Yaskawa INFORM job: DEMO_ROOF_UPPER_0625_3PAINT_8.JBI

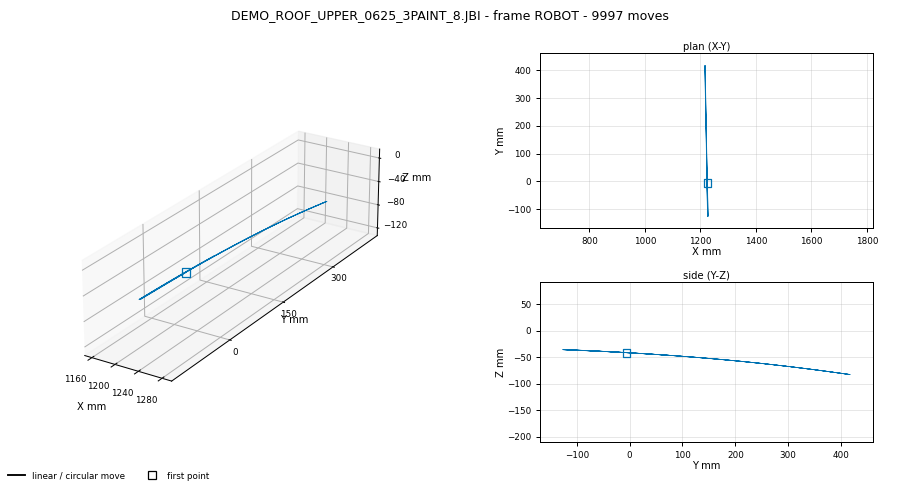
[picture p0: tool path of DEMO_ROOF_UPPER_0625_3PAINT_8.JBI in frame ROBOT, 9997 of 9997 moves have a stored position in this frame; points joined in program order, loops and branches not executed]
/JOB
//NAME DEMO_ROOF_UPPER_0625_3PAINT8
//POS
///NPOS 9997,0,0,0,0,0
///TOOL 0
///USER 0
///POSTYPE ROBOT
///RECTAN
///RCONF 1,0,0,0,0,0,0,0,0,0,0,0,0,0,0,0,0,0,0,0,0,0,0,0
C00000=1225.284,-6.004,-41.147,-179.569,5.363,148.803
C00001=1225.289,-6.253,-41.132,-179.571,5.363,148.804
C00002=1225.293,-6.503,-41.118,-179.574,5.362,148.805
C00003=1225.298,-6.753,-41.104,-179.576,5.362,148.805
C00004=1225.303,-7.002,-41.089,-179.579,5.361,148.806
C00005=1225.308,-7.251,-41.076,-179.581,5.362,148.807
C00006=1225.313,-7.501,-41.063,-179.584,5.361,148.807
C00007=1225.318,-7.751,-41.048,-179.586,5.361,148.808
C00008=1225.323,-8.001,-41.034,-179.588,5.361,148.809
C00009=1225.329,-8.250,-41.020,-179.591,5.360,148.809
C00010=1225.334,-8.500,-41.006,-179.594,5.360,148.810
C00011=1225.339,-8.749,-40.992,-179.596,5.359,148.811
C00012=1225.344,-8.999,-40.977,-179.598,5.360,148.811
C00013=1225.349,-9.248,-40.964,-179.601,5.359,148.812
C00014=1225.354,-9.497,-40.950,-179.604,5.359,148.813
C00015=1225.359,-9.747,-40.935,-179.606,5.359,148.814
C00016=1225.364,-9.997,-40.922,-179.609,5.358,148.814
C00017=1225.369,-10.246,-40.908,-179.611,5.358,148.815
C00018=1225.374,-10.496,-40.894,-179.614,5.357,148.816
C00019=1225.379,-10.746,-40.880,-179.616,5.358,148.816
C00020=1225.384,-10.995,-40.866,-179.619,5.357,148.817
C00021=1225.389,-11.244,-40.852,-179.621,5.357,148.818
C00022=1225.394,-11.495,-40.838,-179.623,5.357,148.818
C00023=1225.400,-11.744,-40.824,-179.625,5.356,148.819
C00024=1225.405,-11.993,-40.810,-179.628,5.356,148.820
C00025=1225.409,-12.243,-40.796,-179.630,5.356,148.820
C00026=1225.414,-12.492,-40.782,-179.633,5.355,148.821
C00027=1225.420,-12.742,-40.769,-179.636,5.355,148.822
C00028=1225.425,-12.992,-40.755,-179.638,5.354,148.822
C00029=1225.429,-13.241,-40.741,-179.640,5.355,148.823
C00030=1225.435,-13.490,-40.727,-179.643,5.354,148.824
C00031=1225.440,-13.741,-40.713,-179.646,5.354,148.824
C00032=1225.445,-13.990,-40.699,-179.648,5.354,148.825
C00033=1225.450,-14.239,-40.686,-179.650,5.353,148.826
C00034=1225.455,-14.489,-40.672,-179.653,5.353,148.826
C00035=1225.460,-14.739,-40.658,-179.655,5.353,148.827
C00036=1225.465,-14.988,-40.644,-179.658,5.353,148.828
C00037=1225.470,-15.237,-40.630,-179.660,5.352,148.829
C00038=1225.475,-15.487,-40.617,-179.663,5.352,148.829
C00039=1225.480,-15.737,-40.603,-179.665,5.352,148.830
C00040=1225.485,-15.986,-40.589,-179.668,5.352,148.831
C00041=1225.490,-16.236,-40.576,-179.670,5.351,148.831
C00042=1225.495,-16.485,-40.562,-179.672,5.351,148.832
C00043=1225.500,-16.735,-40.548,-179.675,5.351,148.833
C00044=1225.506,-16.985,-40.535,-179.678,5.350,148.833
C00045=1225.510,-17.234,-40.521,-179.680,5.351,148.834
C00046=1225.516,-17.484,-40.507,-179.683,5.350,148.835
C00047=1225.521,-17.733,-40.494,-179.685,5.350,148.835
C00048=1225.526,-17.983,-40.480,-179.687,5.350,148.836
C00049=1225.531,-18.233,-40.466,-179.690,5.349,148.837
C00050=1225.536,-18.482,-40.452,-179.693,5.349,148.838
C00051=1225.541,-18.732,-40.439,-179.695,5.350,148.838
C00052=1225.546,-18.981,-40.425,-179.698,5.349,148.839
C00053=1225.551,-19.231,-40.411,-179.700,5.349,148.840
C00054=1225.556,-19.480,-40.398,-179.703,5.349,148.841
C00055=1225.561,-19.730,-40.384,-179.705,5.348,148.841
C00056=1225.567,-19.979,-40.371,-179.708,5.348,148.842
C00057=1225.572,-20.229,-40.357,-179.710,5.348,148.843
C00058=1225.577,-20.479,-40.344,-179.713,5.348,148.843
C00059=1225.582,-20.728,-40.330,-179.715,5.347,148.844
C00060=1225.587,-20.978,-40.317,-179.717,5.347,148.845
C00061=1225.592,-21.227,-40.303,-179.720,5.347,148.845
C00062=1225.597,-21.477,-40.290,-179.723,5.346,148.846
C00063=1225.602,-21.726,-40.276,-179.725,5.346,148.847
C00064=1225.607,-21.977,-40.263,-179.727,5.346,148.848
C00065=1225.612,-22.246,-40.248,-179.730,5.346,148.848
C00066=1225.618,-22.515,-40.233,-179.733,5.345,148.849
C00067=1225.624,-22.784,-40.218,-179.735,5.345,148.850
C00068=1225.629,-23.054,-40.205,-179.738,5.345,148.851
C00069=1225.634,-23.303,-40.191,-179.741,5.345,148.851
C00070=1225.639,-23.553,-40.178,-179.743,5.344,148.852
C00071=1225.645,-23.802,-40.164,-179.745,5.345,148.853
C00072=1225.649,-24.052,-40.151,-179.748,5.344,148.853
C00073=1225.654,-24.302,-40.137,-179.751,5.344,148.854
C00074=1225.659,-24.551,-40.124,-179.753,5.344,148.855
C00075=1225.664,-24.801,-40.110,-179.755,5.344,148.855
C00076=1225.670,-25.050,-40.097,-179.758,5.343,148.856
C00077=1225.674,-25.300,-40.084,-179.760,5.343,148.857
C00078=1225.680,-25.550,-40.070,-179.763,5.343,148.857
C00079=1225.685,-25.799,-40.057,-179.766,5.342,148.858
C00080=1225.690,-26.049,-40.044,-179.768,5.343,148.859
C00081=1225.695,-26.298,-40.030,-179.770,5.342,148.860
C00082=1225.701,-26.548,-40.017,-179.773,5.342,148.860
C00083=1225.705,-26.798,-40.004,-179.775,5.342,148.861
C00084=1225.710,-27.047,-39.990,-179.778,5.342,148.862
C00085=1225.716,-27.296,-39.977,-179.780,5.341,148.862
C00086=1225.720,-27.546,-39.964,-179.782,5.341,148.863
C00087=1225.726,-27.795,-39.950,-179.785,5.341,148.864
C00088=1225.730,-28.045,-39.937,-179.788,5.340,148.864
C00089=1225.736,-28.295,-39.924,-179.790,5.341,148.865
C00090=1225.741,-28.545,-39.911,-179.792,5.340,148.866
C00091=1225.746,-28.794,-39.897,-179.795,5.340,148.867
C00092=1225.751,-29.044,-39.884,-179.797,5.340,148.867
C00093=1225.757,-29.294,-39.871,-179.800,5.339,148.868
C00094=1225.761,-29.543,-39.857,-179.802,5.340,148.869
C00095=1225.766,-29.792,-39.845,-179.805,5.339,148.869
C00096=1225.772,-30.042,-39.832,-179.807,5.339,148.870
C00097=1225.776,-30.292,-39.819,-179.809,5.339,148.871
C00098=1225.782,-30.541,-39.805,-179.812,5.339,148.871
C00099=1225.786,-30.791,-39.792,-179.815,5.338,148.872
C00100=1225.792,-31.040,-39.779,-179.817,5.338,148.873
C00101=1225.797,-31.291,-39.766,-179.819,5.338,148.874
C00102=1225.802,-31.540,-39.753,-179.822,5.337,148.874
C00103=1225.808,-31.789,-39.739,-179.824,5.338,148.875
C00104=1225.812,-32.039,-39.726,-179.827,5.337,148.876
C00105=1225.817,-32.288,-39.714,-179.829,5.338,148.876
C00106=1225.822,-32.539,-39.700,-179.832,5.337,148.877
C00107=1225.828,-32.788,-39.687,-179.834,5.337,148.878
C00108=1225.833,-33.037,-39.675,-179.836,5.337,148.878
C00109=1225.838,-33.287,-39.660,-179.839,5.336,148.879
C00110=1225.843,-33.536,-39.648,-179.842,5.336,148.880
C00111=1225.847,-33.786,-39.635,-179.844,5.336,148.881
C00112=1225.853,-34.036,-39.622,-179.846,5.336,148.881
C00113=1225.858,-34.285,-39.609,-179.848,5.336,148.882
C00114=1225.863,-34.535,-39.596,-179.851,5.336,148.883
C00115=1225.869,-34.785,-39.583,-179.854,5.335,148.883
C00116=1225.874,-35.034,-39.570,-179.856,5.335,148.884
C00117=1225.878,-35.284,-39.557,-179.859,5.335,148.885
C00118=1225.884,-35.533,-39.543,-179.861,5.334,148.885
C00119=1225.888,-35.783,-39.530,-179.863,5.335,148.886
C00120=1225.893,-36.033,-39.518,-179.866,5.334,148.887
C00121=1225.899,-36.282,-39.505,-179.869,5.334,148.888
C00122=1225.904,-36.532,-39.492,-179.871,5.334,148.888
C00123=1225.909,-36.782,-39.479,-179.873,5.334,148.889
C00124=1225.914,-37.031,-39.467,-179.875,5.334,148.890
C00125=1225.919,-37.281,-39.453,-179.878,5.333,148.890
C00126=1225.924,-37.531,-39.440,-179.881,5.333,148.891
C00127=1225.930,-37.780,-39.428,-179.883,5.333,148.892
C00128=1225.934,-38.030,-39.415,-179.885,5.333,148.892
C00129=1225.940,-38.280,-39.402,-179.888,5.333,148.893
C00130=1225.945,-38.529,-39.389,-179.890,5.333,148.894
C00131=1225.950,-38.779,-39.376,-179.893,5.332,148.895
C00132=1225.955,-39.028,-39.363,-179.895,5.332,148.895
C00133=1225.961,-39.278,-39.350,-179.898,5.332,148.896
C00134=1225.966,-39.527,-39.338,-179.900,5.331,148.897
C00135=1225.970,-39.777,-39.325,-179.902,5.332,148.897
C00136=1225.975,-40.026,-39.312,-179.905,5.331,148.898
C00137=1225.981,-40.276,-39.299,-179.907,5.332,148.899
C00138=1225.986,-40.526,-39.286,-179.910,5.331,148.899
C00139=1225.991,-40.775,-39.273,-179.912,5.331,148.900
C00140=1225.996,-41.025,-39.261,-179.915,5.331,148.901
C00141=1226.001,-41.275,-39.248,-179.917,5.330,148.902
C00142=1226.006,-41.525,-39.236,-179.919,5.331,148.902
C00143=1226.011,-41.774,-39.223,-179.922,5.330,148.903
C00144=1226.017,-42.024,-39.210,-179.925,5.330,148.904
C00145=1226.021,-42.274,-39.197,-179.927,5.330,148.904
C00146=1226.027,-42.523,-39.184,-179.929,5.330,148.905
C00147=1226.032,-42.772,-39.172,-179.931,5.330,148.906
C00148=1226.037,-43.022,-39.159,-179.934,5.329,148.906
C00149=1226.041,-43.272,-39.146,-179.937,5.329,148.907
C00150=1226.047,-43.522,-39.134,-179.939,5.329,148.908
C00151=1226.053,-43.771,-39.121,-179.942,5.329,148.909
C00152=1226.058,-44.020,-39.109,-179.944,5.328,148.909
C00153=1226.062,-44.271,-39.096,-179.946,5.329,148.910
C00154=1226.067,-44.520,-39.083,-179.949,5.328,148.911
C00155=1226.073,-44.769,-39.070,-179.951,5.329,148.911
C00156=1226.078,-45.019,-39.059,-179.954,5.328,148.912
C00157=1226.083,-45.269,-39.046,-179.956,5.328,148.913
C00158=1226.088,-45.518,-39.033,-179.958,5.328,148.913
C00159=1226.093,-45.768,-39.020,-179.961,5.327,148.914
C00160=1226.099,-46.017,-39.007,-179.963,5.328,148.915
C00161=1226.104,-46.267,-38.995,-179.966,5.327,148.916
C00162=1226.109,-46.517,-38.982,-179.968,5.328,148.916
C00163=1226.114,-46.767,-38.970,-179.971,5.327,148.917
C00164=1226.119,-47.016,-38.957,-179.973,5.327,148.918
C00165=1226.124,-47.266,-38.945,-179.975,5.327,148.918
C00166=1226.129,-47.515,-38.933,-179.978,5.326,148.919
C00167=1226.134,-47.765,-38.920,-179.980,5.327,148.920
C00168=1226.139,-48.015,-38.907,-179.983,5.326,148.920
C00169=1226.145,-48.284,-38.895,-179.986,5.326,148.921
C00170=1226.151,-48.554,-38.880,-179.988,5.327,148.922
C00171=1226.156,-48.825,-38.867,-179.991,5.326,148.923
C00172=1226.162,-49.094,-38.854,-179.993,5.326,148.923
C00173=1226.166,-49.344,-38.841,-179.996,5.325,148.924
C00174=1226.172,-49.594,-38.829,-179.998,5.325,148.925
C00175=1226.177,-49.843,-38.817,179.999,5.325,148.926
C00176=1226.182,-50.092,-38.804,179.997,5.325,148.926
C00177=1226.187,-50.342,-38.792,179.994,5.325,148.927
C00178=1226.192,-50.591,-38.779,179.992,5.325,148.928
C00179=1226.197,-50.841,-38.766,179.990,5.325,148.928
C00180=1226.202,-51.091,-38.755,179.987,5.324,148.929
C00181=1226.207,-51.341,-38.742,179.985,5.324,148.930
C00182=1226.213,-51.590,-38.729,179.982,5.324,148.931
C00183=1226.218,-51.840,-38.717,179.980,5.324,148.931
C00184=1226.223,-52.089,-38.705,179.978,5.324,148.932
C00185=1226.229,-52.339,-38.693,179.975,5.323,148.933
C00186=1226.234,-52.589,-38.680,179.973,5.324,148.933
C00187=1226.238,-52.839,-38.667,179.970,5.323,148.934
C00188=1226.244,-53.089,-38.656,179.968,5.324,148.935
C00189=1226.249,-53.338,-38.643,179.965,5.323,148.935
C00190=1226.254,-53.588,-38.631,179.963,5.323,148.936
C00191=1226.259,-53.837,-38.619,179.961,5.323,148.937
C00192=1226.264,-54.087,-38.607,179.958,5.322,148.938
C00193=1226.269,-54.336,-38.595,179.956,5.323,148.938
C00194=1226.275,-54.586,-38.583,179.953,5.322,148.939
C00195=1226.279,-54.836,-38.570,179.951,5.323,148.940
C00196=1226.284,-55.086,-38.558,179.948,5.322,148.940
C00197=1226.290,-55.335,-38.545,179.946,5.322,148.941
C00198=1226.295,-55.585,-38.533,179.944,5.322,148.942
C00199=1226.300,-55.834,-38.521,179.941,5.322,148.942
C00200=1226.305,-56.084,-38.509,179.939,5.322,148.943
C00201=1226.310,-56.333,-38.497,179.936,5.321,148.944
C00202=1226.315,-56.583,-38.485,179.934,5.322,148.945
C00203=1226.321,-56.833,-38.472,179.932,5.321,148.945
C00204=1226.326,-57.083,-38.460,179.929,5.322,148.946
C00205=1226.331,-57.332,-38.448,179.927,5.321,148.947
C00206=1226.336,-57.582,-38.437,179.924,5.321,148.947
C00207=1226.341,-57.831,-38.424,179.922,5.321,148.948
C00208=1226.346,-58.081,-38.412,179.919,5.321,148.949
C00209=1226.351,-58.331,-38.399,179.917,5.321,148.950
C00210=1226.356,-58.581,-38.387,179.915,5.320,148.950
C00211=1226.362,-58.831,-38.375,179.913,5.321,148.951
C00212=1226.366,-59.080,-38.363,179.910,5.320,148.952
C00213=1226.372,-59.330,-38.351,179.908,5.321,148.952
C00214=1226.377,-59.579,-38.339,179.905,5.320,148.953
C00215=1226.382,-59.829,-38.327,179.902,5.320,148.954
C00216=1226.388,-60.079,-38.315,179.900,5.320,148.954
C00217=1226.392,-60.328,-38.303,179.898,5.320,148.955
C00218=1226.397,-60.578,-38.291,179.896,5.320,148.956
C00219=1226.403,-60.828,-38.279,179.893,5.319,148.957
C00220=1226.408,-61.077,-38.267,179.891,5.320,148.957
C00221=1226.413,-61.327,-38.255,179.888,5.319,148.958
C00222=1226.418,-61.577,-38.244,179.885,5.319,148.959
C00223=1226.423,-61.826,-38.231,179.883,5.319,148.959
C00224=1226.429,-62.076,-38.219,179.881,5.319,148.960
C00225=1226.433,-62.325,-38.208,179.879,5.319,148.961
C00226=1226.438,-62.575,-38.195,179.876,5.319,148.962
C00227=1226.444,-62.825,-38.183,179.874,5.319,148.962
C00228=1226.449,-63.075,-38.171,179.871,5.318,148.963
C00229=1226.454,-63.324,-38.160,179.869,5.319,148.964
C00230=1226.459,-63.574,-38.148,179.866,5.318,148.964
C00231=1226.464,-63.824,-38.136,179.864,5.318,148.965
C00232=1226.469,-64.073,-38.124,179.862,5.318,148.966
C00233=1226.474,-64.322,-38.112,179.859,5.318,148.966
C00234=1226.480,-64.572,-38.100,179.857,5.318,148.967
C00235=1226.485,-64.822,-38.088,179.854,5.318,148.968
C00236=1226.490,-65.072,-38.077,179.852,5.318,148.969
C00237=1226.495,-65.322,-38.065,179.850,5.317,148.969
C00238=1226.501,-65.571,-38.053,179.847,5.318,148.970
C00239=1226.506,-65.820,-38.041,179.845,5.317,148.971
C00240=1226.511,-66.070,-38.029,179.843,5.318,148.971
C00241=1226.517,-66.320,-38.017,179.840,5.317,148.972
C00242=1226.521,-66.570,-38.006,179.837,5.317,148.973
C00243=1226.526,-66.819,-37.994,179.835,5.317,148.974
C00244=1226.532,-67.069,-37.982,179.833,5.317,148.974
C00245=1226.536,-67.319,-37.970,179.830,5.317,148.975
C00246=1226.542,-67.568,-37.959,179.828,5.316,148.976
C00247=1226.547,-67.818,-37.947,179.826,5.317,148.976
C00248=1226.552,-68.068,-37.935,179.823,5.316,148.977
C00249=1226.557,-68.317,-37.923,179.821,5.317,148.978
C00250=1226.562,-68.567,-37.911,179.818,5.316,148.978
C00251=1226.568,-68.816,-37.900,179.816,5.317,148.979
C00252=1226.573,-69.066,-37.888,179.814,5.316,148.980
C00253=1226.578,-69.316,-37.877,179.811,5.316,148.981
C00254=1226.583,-69.566,-37.865,179.809,5.316,148.981
C00255=1226.588,-69.815,-37.854,179.806,5.315,148.982
C00256=1226.594,-70.065,-37.842,179.804,5.316,148.983
C00257=1226.599,-70.315,-37.830,179.801,5.315,148.983
C00258=1226.604,-70.565,-37.819,179.799,5.316,148.984
C00259=1226.609,-70.814,-37.806,179.797,5.315,148.985
C00260=1226.614,-71.063,-37.795,179.795,5.316,148.986
C00261=1226.620,-71.313,-37.783,179.792,5.315,148.986
C00262=1226.624,-71.563,-37.772,179.790,5.315,148.987
C00263=1226.630,-71.813,-37.760,179.787,5.315,148.988
C00264=1226.634,-72.062,-37.749,179.785,5.315,148.988
C00265=1226.640,-72.312,-37.737,179.782,5.315,148.989
C00266=1226.645,-72.562,-37.725,179.780,5.315,148.990
C00267=1226.650,-72.811,-37.714,179.778,5.315,148.991
C00268=1226.656,-73.061,-37.702,179.775,5.314,148.991
C00269=1226.661,-73.311,-37.691,179.773,5.315,148.992
C00270=1226.666,-73.561,-37.679,179.770,5.314,148.993
C00271=1226.671,-73.810,-37.668,179.768,5.315,148.993
C00272=1226.676,-74.060,-37.656,179.765,5.314,148.994
C00273=1226.682,-74.330,-37.644,179.763,5.314,148.995
C00274=1226.688,-74.601,-37.631,179.761,5.314,148.995
C00275=1226.693,-74.871,-37.620,179.758,5.314,148.996
C00276=1226.698,-75.141,-37.607,179.755,5.314,148.997
C00277=1226.704,-75.391,-37.595,179.753,5.314,148.998
C00278=1226.709,-75.641,-37.583,179.751,5.314,148.999
C00279=1226.714,-75.891,-37.572,179.748,5.314,148.999
C00280=1226.719,-76.139,-37.561,179.746,5.314,149.000
C00281=1226.725,-76.390,-37.549,179.743,5.314,149.001
C00282=1226.730,-76.640,-37.538,179.741,5.314,149.001
C00283=1226.735,-76.890,-37.526,179.738,5.313,149.002
C00284=1226.740,-77.138,-37.515,179.736,5.314,149.003
C00285=1226.746,-77.388,-37.503,179.734,5.313,149.003
C00286=1226.751,-77.638,-37.492,179.732,5.313,149.004
C00287=1226.755,-77.888,-37.481,179.729,5.313,149.005
C00288=1226.761,-78.138,-37.469,179.727,5.312,149.005
C00289=1226.766,-78.387,-37.458,179.725,5.313,149.006
C00290=1226.772,-78.637,-37.447,179.722,5.312,149.007
C00291=1226.776,-78.887,-37.436,179.720,5.313,149.008
C00292=1226.782,-79.137,-37.424,179.717,5.312,149.008
C00293=1226.787,-79.386,-37.413,179.715,5.313,149.009
C00294=1226.792,-79.635,-37.402,179.712,5.312,149.010
C00295=1226.798,-79.886,-37.390,179.710,5.312,149.010
C00296=1226.802,-80.135,-37.379,179.708,5.312,149.011
C00297=1226.808,-80.384,-37.368,179.706,5.312,149.012
C00298=1226.813,-80.634,-37.356,179.703,5.312,149.012
C00299=1226.818,-80.884,-37.345,179.701,5.312,149.013
C00300=1226.823,-81.134,-37.334,179.698,5.312,149.014
C00301=1226.829,-81.383,-37.323,179.696,5.312,149.015
C00302=1226.833,-81.633,-37.312,179.693,5.312,149.015
C00303=1226.839,-81.883,-37.300,179.691,5.312,149.016
C00304=1226.844,-82.133,-37.289,179.689,5.312,149.017
C00305=1226.849,-82.382,-37.278,179.687,5.312,149.017
C00306=1226.855,-82.632,-37.266,179.684,5.311,149.018
C00307=1226.859,-82.882,-37.255,179.682,5.312,149.019
C00308=1226.864,-83.132,-37.244,179.679,5.311,149.020
C00309=1226.870,-83.381,-37.233,179.677,5.312,149.020
C00310=1226.875,-83.631,-37.222,179.674,5.311,149.021
C00311=1226.880,-83.880,-37.210,179.672,5.312,149.022
C00312=1226.885,-84.130,-37.200,179.670,5.311,149.022
C00313=1226.891,-84.380,-37.188,179.667,5.312,149.023
C00314=1226.895,-84.629,-37.177,179.665,5.311,149.024
C00315=1226.901,-84.879,-37.167,179.663,5.311,149.024
C00316=1226.906,-85.129,-37.155,179.661,5.311,149.025
C00317=1226.911,-85.379,-37.144,179.658,5.311,149.026
C00318=1226.916,-85.629,-37.133,179.656,5.311,149.026
C00319=1226.921,-85.878,-37.122,179.654,5.311,149.027
C00320=1226.927,-86.128,-37.110,179.651,5.310,149.028
C00321=1226.932,-86.378,-37.100,179.649,5.311,149.029
C00322=1226.937,-86.627,-37.089,179.646,5.310,149.029
C00323=1226.942,-86.877,-37.078,179.644,5.311,149.030
C00324=1226.948,-87.127,-37.066,179.641,5.310,149.031
C00325=1226.953,-87.376,-37.055,179.639,5.311,149.031
C00326=1226.958,-87.626,-37.045,179.637,5.310,149.032
C00327=1226.963,-87.876,-37.033,179.635,5.310,149.033
C00328=1226.969,-88.126,-37.023,179.632,5.310,149.034
C00329=1226.974,-88.375,-37.011,179.630,5.310,149.034
C00330=1226.979,-88.624,-37.000,179.627,5.310,149.035
C00331=1226.984,-88.874,-36.990,179.625,5.310,149.036
C00332=1226.989,-89.124,-36.979,179.622,5.310,149.036
C00333=1226.995,-89.374,-36.968,179.620,5.310,149.037
C00334=1227.000,-89.624,-36.956,179.618,5.310,149.038
C00335=1227.005,-89.874,-36.946,179.616,5.310,149.038
C00336=1227.010,-90.123,-36.935,179.613,5.309,149.039
C00337=1227.015,-90.373,-36.924,179.611,5.310,149.040
C00338=1227.021,-90.622,-36.913,179.609,5.309,149.040
C00339=1227.026,-90.872,-36.902,179.607,5.310,149.041
C00340=1227.031,-91.122,-36.891,179.604,5.309,149.042
C00341=1227.036,-91.372,-36.881,179.602,5.309,149.043
C00342=1227.041,-91.621,-36.870,179.599,5.309,149.043
C00343=1227.046,-91.871,-36.859,179.597,5.309,149.044
C00344=1227.051,-92.120,-36.848,179.594,5.309,149.045
C00345=1227.057,-92.371,-36.837,179.592,5.309,149.045
C00346=1227.062,-92.620,-36.826,179.590,5.309,149.046
C00347=1227.067,-92.870,-36.815,179.587,5.309,149.047
C00348=1227.072,-93.119,-36.804,179.585,5.309,149.048
C00349=1227.077,-93.369,-36.794,179.583,5.309,149.048
C00350=1227.082,-93.619,-36.783,179.580,5.309,149.049
C00351=1227.088,-93.869,-36.772,179.578,5.309,149.050
C00352=1227.093,-94.119,-36.762,179.576,5.308,149.050
C00353=1227.099,-94.368,-36.750,179.574,5.309,149.051
C00354=1227.104,-94.618,-36.740,179.571,5.308,149.052
C00355=1227.109,-94.867,-36.729,179.569,5.309,149.052
C00356=1227.114,-95.117,-36.718,179.566,5.308,149.053
C00357=1227.120,-95.367,-36.708,179.564,5.308,149.054
C00358=1227.124,-95.617,-36.697,179.561,5.308,149.054
C00359=1227.129,-95.867,-36.686,179.559,5.308,149.055
C00360=1227.135,-96.116,-36.675,179.557,5.308,149.056
C00361=1227.140,-96.366,-36.665,179.555,5.308,149.057
C00362=1227.145,-96.616,-36.654,179.552,5.308,149.057
C00363=1227.150,-96.865,-36.643,179.550,5.308,149.058
C00364=1227.156,-97.115,-36.633,179.547,5.308,149.059
C00365=1227.161,-97.365,-36.622,179.545,5.308,149.059
C00366=1227.166,-97.614,-36.611,179.543,5.307,149.060
C00367=1227.172,-97.864,-36.600,179.541,5.308,149.061
C00368=1227.177,-98.114,-36.590,179.538,5.307,149.061
C00369=1227.182,-98.364,-36.579,179.536,5.308,149.062
C00370=1227.187,-98.613,-36.569,179.534,5.308,149.063
C00371=1227.192,-98.863,-36.558,179.531,5.307,149.063
C00372=1227.198,-99.113,-36.548,179.529,5.308,149.064
C00373=1227.203,-99.363,-36.536,179.526,5.307,149.065
C00374=1227.208,-99.612,-36.526,179.524,5.308,149.066
C00375=1227.213,-99.862,-36.516,179.522,5.307,149.066
C00376=1227.219,-100.111,-36.505,179.520,5.308,149.067
C00377=1227.224,-100.383,-36.494,179.517,5.307,149.068
C00378=1227.230,-100.654,-36.482,179.514,5.307,149.068
C00379=1227.235,-100.924,-36.471,179.512,5.307,149.069
C00380=1227.241,-101.196,-36.459,179.509,5.307,149.070
C00381=1227.247,-101.445,-36.449,179.507,5.307,149.071
C00382=1227.251,-101.695,-36.438,179.505,5.307,149.071
C00383=1227.257,-101.944,-36.428,179.503,5.307,149.072
C00384=1227.262,-102.195,-36.417,179.500,5.307,149.073
C00385=1227.267,-102.444,-36.408,179.498,5.307,149.073
C00386=1227.272,-102.694,-36.397,179.495,5.307,149.074
C00387=1227.277,-102.943,-36.386,179.493,5.307,149.075
C00388=1227.282,-103.193,-36.376,179.490,5.306,149.076
C00389=1227.288,-103.443,-36.365,179.488,5.307,149.076
C00390=1227.293,-103.693,-36.355,179.486,5.306,149.077
C00391=1227.298,-103.943,-36.345,179.484,5.306,149.078
C00392=1227.304,-104.192,-36.334,179.482,5.307,149.078
C00393=1227.309,-104.442,-36.324,179.479,5.306,149.079
C00394=1227.314,-104.691,-36.313,179.477,5.307,149.080
C00395=1227.319,-104.942,-36.302,179.474,5.306,149.080
C00396=1227.324,-105.191,-36.293,179.472,5.307,149.081
C00397=1227.329,-105.441,-36.282,179.470,5.306,149.082
C00398=1227.335,-105.691,-36.272,179.468,5.307,149.083
C00399=1227.340,-105.940,-36.262,179.465,5.306,149.083
C00400=1227.345,-106.190,-36.251,179.463,5.306,149.084
C00401=1227.351,-106.440,-36.241,179.461,5.306,149.084
C00402=1227.356,-106.690,-36.230,179.459,5.306,149.085
C00403=1227.361,-106.940,-36.220,179.456,5.306,149.086
C00404=1227.366,-107.188,-36.210,179.454,5.306,149.087
C00405=1227.371,-107.439,-36.199,179.451,5.306,149.087
C00406=1227.377,-107.688,-36.189,179.449,5.306,149.088
C00407=1227.382,-107.938,-36.178,179.446,5.305,149.089
C00408=1227.387,-108.188,-36.168,179.444,5.306,149.089
C00409=1227.393,-108.437,-36.158,179.442,5.306,149.090
C00410=1227.397,-108.687,-36.148,179.440,5.305,149.091
C00411=1227.403,-108.937,-36.138,179.438,5.306,149.091
C00412=1227.408,-109.187,-36.128,179.435,5.305,149.092
C00413=1227.413,-109.437,-36.117,179.433,5.306,149.093
C00414=1227.419,-109.686,-36.107,179.430,5.305,149.094
C00415=1227.423,-109.936,-36.097,179.428,5.306,149.094
C00416=1227.429,-110.186,-36.087,179.426,5.305,149.095
C00417=1227.434,-110.435,-36.076,179.424,5.306,149.096
C00418=1227.439,-110.686,-36.066,179.421,5.305,149.096
C00419=1227.445,-110.935,-36.056,179.419,5.305,149.097
C00420=1227.450,-111.184,-36.046,179.417,5.305,149.098
C00421=1227.455,-111.435,-36.035,179.415,5.305,149.098
C00422=1227.460,-111.684,-36.025,179.412,5.305,149.099
C00423=1227.466,-111.934,-36.015,179.410,5.305,149.100
C00424=1227.471,-112.184,-36.006,179.408,5.305,149.100
C00425=1227.476,-112.434,-35.996,179.405,5.305,149.101
C00426=1227.482,-112.683,-35.985,179.403,5.305,149.102
C00427=1227.487,-112.934,-35.975,179.400,5.305,149.103
C00428=1227.492,-113.183,-35.965,179.399,5.305,149.103
C00429=1227.497,-113.432,-35.955,179.396,5.304,149.104
C00430=1227.502,-113.683,-35.944,179.394,5.305,149.104
C00431=1227.508,-113.932,-35.934,179.391,5.304,149.105
C00432=1227.513,-114.181,-35.925,179.389,5.305,149.106
C00433=1227.518,-114.431,-35.914,179.386,5.304,149.107
C00434=1227.524,-114.682,-35.904,179.384,5.305,149.107
C00435=1227.528,-114.931,-35.895,179.382,5.305,149.108
C00436=1227.534,-115.181,-35.885,179.380,5.304,149.109
C00437=1227.539,-115.431,-35.874,179.378,5.305,149.109
C00438=1227.544,-115.680,-35.864,179.375,5.304,149.110
C00439=1227.549,-115.930,-35.854,179.373,5.305,149.111
C00440=1227.555,-116.180,-35.845,179.370,5.304,149.111
C00441=1227.560,-116.430,-35.835,179.368,5.305,149.112
C00442=1227.565,-116.679,-35.825,179.366,5.304,149.113
C00443=1227.571,-116.929,-35.814,179.364,5.304,149.113
C00444=1227.576,-117.178,-35.805,179.361,5.304,149.114
C00445=1227.581,-117.429,-35.795,179.359,5.304,149.115
C00446=1227.587,-117.678,-35.785,179.357,5.304,149.115
C00447=1227.591,-117.928,-35.775,179.355,5.304,149.116
C00448=1227.596,-118.178,-35.764,179.352,5.304,149.117
C00449=1227.602,-118.427,-35.754,179.350,5.304,149.118
C00450=1227.607,-118.677,-35.745,179.348,5.304,149.118
C00451=1227.613,-118.927,-35.735,179.346,5.304,149.119
C00452=1227.618,-119.176,-35.725,179.343,5.304,149.120
C00453=1227.623,-119.426,-35.715,179.341,5.304,149.120
C00454=1227.629,-119.676,-35.705,179.339,5.304,149.121
C00455=1227.633,-119.926,-35.696,179.336,5.303,149.122
C00456=1227.639,-120.175,-35.686,179.334,5.304,149.122
C00457=1227.644,-120.426,-35.676,179.332,5.304,149.123
C00458=1227.649,-120.675,-35.666,179.330,5.303,149.124
C00459=1227.655,-120.925,-35.656,179.328,5.304,149.124
C00460=1227.660,-121.174,-35.646,179.325,5.303,149.125
C00461=1227.666,-121.424,-35.637,179.323,5.304,149.126
C00462=1227.670,-121.674,-35.627,179.320,5.303,149.126
C00463=1227.675,-121.924,-35.617,179.318,5.304,149.127
C00464=1227.681,-122.174,-35.607,179.316,5.303,149.128
C00465=1227.686,-122.423,-35.598,179.314,5.303,149.128
C00466=1227.691,-122.673,-35.587,179.312,5.304,149.129
C00467=1227.696,-122.923,-35.578,179.309,5.303,149.130
C00468=1227.702,-123.173,-35.568,179.307,5.304,149.131
C00469=1227.707,-123.422,-35.558,179.304,5.303,149.131
C00470=1227.713,-123.672,-35.549,179.303,5.303,149.132
C00471=1227.718,-123.921,-35.539,179.300,5.303,149.132
C00472=1227.723,-124.172,-35.529,179.298,5.303,149.133
C00473=1227.728,-124.421,-35.520,179.295,5.303,149.134
C00474=1227.733,-124.671,-35.509,179.293,5.303,149.135
C00475=1227.739,-124.921,-35.501,179.290,5.303,149.135
C00476=1227.744,-125.170,-35.490,179.289,5.303,149.136
C00477=1227.749,-125.420,-35.481,179.287,5.303,149.137
C00478=1227.754,-125.671,-35.471,179.284,5.303,149.137
C00479=1227.759,-125.920,-35.462,179.282,5.303,149.138
C00480=1227.765,-126.170,-35.452,179.279,5.303,149.139
C00481=1227.343,-126.181,-35.488,179.275,5.306,149.141
C00482=1227.338,-125.931,-35.497,179.277,5.307,149.140
C00483=1227.333,-125.681,-35.507,179.279,5.306,149.139
C00484=1227.328,-125.431,-35.517,179.282,5.307,149.139
C00485=1227.322,-125.181,-35.527,179.284,5.306,149.138
C00486=1227.317,-124.932,-35.536,179.286,5.306,149.137
C00487=1227.312,-124.682,-35.546,179.289,5.306,149.137
C00488=1227.307,-124.433,-35.555,179.291,5.306,149.136
C00489=1227.301,-124.182,-35.565,179.293,5.307,149.135
C00490=1227.296,-123.933,-35.575,179.295,5.306,149.135
C00491=1227.291,-123.683,-35.585,179.298,5.307,149.134
C00492=1227.286,-123.433,-35.594,179.300,5.306,149.133
C00493=1227.280,-123.184,-35.604,179.303,5.307,149.132
C00494=1227.275,-122.934,-35.613,179.304,5.307,149.132
C00495=1227.269,-122.684,-35.623,179.307,5.306,149.131
C00496=1227.264,-122.434,-35.634,179.309,5.307,149.131
C00497=1227.259,-122.184,-35.643,179.311,5.306,149.130
C00498=1227.254,-121.934,-35.653,179.314,5.307,149.129
C00499=1227.249,-121.685,-35.663,179.316,5.306,149.128
C00500=1227.243,-121.435,-35.672,179.318,5.307,149.128
C00501=1227.239,-121.185,-35.682,179.320,5.307,149.127
C00502=1227.233,-120.936,-35.692,179.323,5.307,149.126
C00503=1227.228,-120.686,-35.701,179.325,5.307,149.126
C00504=1227.222,-120.436,-35.711,179.328,5.307,149.125
C00505=1227.217,-120.187,-35.722,179.330,5.307,149.124
C00506=1227.212,-119.937,-35.732,179.332,5.307,149.124
C00507=1227.207,-119.687,-35.741,179.334,5.307,149.123
C00508=1227.202,-119.437,-35.751,179.336,5.307,149.122
C00509=1227.196,-119.188,-35.761,179.339,5.307,149.122
C00510=1227.191,-118.937,-35.771,179.341,5.307,149.121
C00511=1227.186,-118.688,-35.780,179.344,5.308,149.120
C00512=1227.180,-118.438,-35.791,179.346,5.307,149.120
C00513=1227.175,-118.189,-35.801,179.349,5.308,149.119
C00514=1227.170,-117.938,-35.810,179.350,5.308,149.118
C00515=1227.165,-117.689,-35.820,179.352,5.307,149.118
C00516=1227.160,-117.439,-35.830,179.355,5.308,149.117
C00517=1227.154,-117.190,-35.840,179.357,5.307,149.116
C00518=1227.149,-116.939,-35.851,179.360,5.308,149.115
C00519=1227.144,-116.690,-35.860,179.362,5.307,149.115
C00520=1227.138,-116.440,-35.870,179.364,5.308,149.114
C00521=1227.133,-116.191,-35.880,179.366,5.308,149.114
C00522=1227.128,-115.941,-35.890,179.369,5.308,149.113
C00523=1227.123,-115.691,-35.900,179.371,5.308,149.112
C00524=1227.117,-115.441,-35.910,179.373,5.308,149.111
C00525=1227.113,-115.191,-35.920,179.376,5.308,149.111
C00526=1227.107,-114.941,-35.930,179.378,5.308,149.110
C00527=1227.101,-114.692,-35.940,179.380,5.308,149.109
C00528=1227.097,-114.443,-35.950,179.382,5.308,149.109
C00529=1227.092,-114.192,-35.960,179.385,5.308,149.108
C00530=1227.086,-113.943,-35.970,179.387,5.308,149.107
C00531=1227.080,-113.693,-35.980,179.389,5.308,149.107
C00532=1227.076,-113.443,-35.990,179.391,5.308,149.106
C00533=1227.070,-113.193,-36.000,179.394,5.308,149.105
C00534=1227.065,-112.944,-36.010,179.396,5.308,149.104
C00535=1227.060,-112.693,-36.021,179.399,5.308,149.104
C00536=1227.055,-112.444,-36.031,179.401,5.309,149.103
C00537=1227.049,-112.195,-36.041,179.403,5.309,149.103
C00538=1227.044,-111.945,-36.051,179.405,5.309,149.102
C00539=1227.039,-111.695,-36.062,179.407,5.308,149.101
C00540=1227.034,-111.446,-36.071,179.410,5.309,149.100
C00541=1227.028,-111.196,-36.081,179.412,5.308,149.100
C00542=1227.023,-110.946,-36.092,179.415,5.309,149.099
C00543=1227.018,-110.696,-36.102,179.417,5.308,149.098
C00544=1227.012,-110.446,-36.111,179.420,5.309,149.098
C00545=1227.007,-110.196,-36.122,179.421,5.309,149.097
C00546=1227.002,-109.947,-36.132,179.424,5.309,149.096
C00547=1226.997,-109.696,-36.142,179.426,5.309,149.096
C00548=1226.991,-109.447,-36.153,179.429,5.309,149.095
C00549=1226.986,-109.198,-36.162,179.431,5.309,149.094
C00550=1226.981,-108.947,-36.173,179.433,5.309,149.093
C00551=1226.976,-108.698,-36.183,179.436,5.309,149.093
C00552=1226.970,-108.448,-36.193,179.438,5.309,149.092
C00553=1226.965,-108.198,-36.204,179.440,5.309,149.092
C00554=1226.961,-107.949,-36.214,179.442,5.309,149.091
C00555=1226.955,-107.700,-36.224,179.445,5.309,149.090
C00556=1226.950,-107.450,-36.235,179.447,5.309,149.089
C00557=1226.944,-107.200,-36.245,179.449,5.309,149.089
C00558=1226.939,-106.950,-36.256,179.451,5.309,149.088
C00559=1226.934,-106.700,-36.266,179.454,5.310,149.087
C00560=1226.929,-106.451,-36.276,179.456,5.309,149.087
C00561=1226.924,-106.201,-36.286,179.459,5.310,149.086
C00562=1226.918,-105.951,-36.296,179.461,5.309,149.085
C00563=1226.913,-105.701,-36.307,179.463,5.310,149.085
C00564=1226.908,-105.452,-36.317,179.465,5.310,149.084
C00565=1226.902,-105.202,-36.327,179.468,5.310,149.083
C00566=1226.897,-104.952,-36.338,179.470,5.310,149.083
C00567=1226.892,-104.703,-36.349,179.473,5.310,149.082
C00568=1226.888,-104.453,-36.359,179.475,5.310,149.081
C00569=1226.882,-104.203,-36.369,179.477,5.310,149.080
C00570=1226.877,-103.953,-36.380,179.480,5.310,149.080
C00571=1226.871,-103.704,-36.390,179.482,5.310,149.079
C00572=1226.866,-103.454,-36.400,179.484,5.310,149.078
C00573=1226.861,-103.204,-36.411,179.486,5.310,149.078
C00574=1226.856,-102.955,-36.421,179.489,5.310,149.077
C00575=1226.851,-102.705,-36.432,179.491,5.310,149.076
C00576=1226.845,-102.455,-36.442,179.493,5.310,149.076
C00577=1226.840,-102.205,-36.453,179.495,5.310,149.075
C00578=1226.834,-101.955,-36.463,179.498,5.311,149.074
C00579=1226.830,-101.706,-36.474,179.500,5.310,149.073
C00580=1226.824,-101.456,-36.485,179.503,5.311,149.073
C00581=1226.820,-101.206,-36.495,179.505,5.310,149.072
C00582=1226.813,-100.935,-36.506,179.508,5.311,149.071
C00583=1226.808,-100.664,-36.518,179.510,5.310,149.071
C00584=1226.802,-100.393,-36.529,179.512,5.311,149.070
C00585=1226.796,-100.122,-36.540,179.515,5.311,149.069
C00586=1226.791,-99.872,-36.551,179.517,5.311,149.068
C00587=1226.786,-99.623,-36.562,179.520,5.311,149.068
C00588=1226.781,-99.373,-36.572,179.522,5.311,149.067
C00589=1226.775,-99.124,-36.583,179.525,5.311,149.066
C00590=1226.770,-98.874,-36.594,179.527,5.311,149.066
C00591=1226.765,-98.624,-36.604,179.529,5.311,149.065
C00592=1226.760,-98.374,-36.614,179.532,5.311,149.064
C00593=1226.754,-98.125,-36.625,179.534,5.311,149.063
C00594=1226.749,-97.875,-36.636,179.536,5.311,149.063
C00595=1226.744,-97.625,-36.646,179.538,5.311,149.062
C00596=1226.739,-97.375,-36.657,179.541,5.312,149.062
C00597=1226.734,-97.126,-36.668,179.543,5.311,149.061
C00598=1226.729,-96.876,-36.678,179.545,5.312,149.060
C00599=1226.723,-96.627,-36.689,179.547,5.311,149.059
C00600=1226.718,-96.376,-36.700,179.550,5.312,149.059
C00601=1226.713,-96.127,-36.710,179.552,5.311,149.058
C00602=1226.708,-95.877,-36.721,179.555,5.312,149.057
C00603=1226.703,-95.627,-36.732,179.557,5.311,149.057
C00604=1226.697,-95.377,-36.742,179.560,5.312,149.056
C00605=1226.693,-95.128,-36.753,179.562,5.312,149.055
C00606=1226.687,-94.878,-36.763,179.564,5.312,149.054
C00607=1226.682,-94.629,-36.775,179.567,5.312,149.054
C00608=1226.676,-94.379,-36.786,179.569,5.312,149.053
C00609=1226.671,-94.129,-36.796,179.571,5.312,149.052
C00610=1226.666,-93.880,-36.807,179.573,5.313,149.052
C00611=1226.661,-93.629,-36.818,179.576,5.312,149.051
C00612=1226.656,-93.380,-36.829,179.578,5.313,149.050
C00613=1226.651,-93.130,-36.839,179.580,5.312,149.050
C00614=1226.646,-92.880,-36.850,179.583,5.313,149.049
C00615=1226.640,-92.631,-36.861,179.585,5.312,149.048
C00616=1226.635,-92.381,-36.871,179.588,5.313,149.048
C00617=1226.629,-92.132,-36.883,179.590,5.312,149.047
C00618=1226.624,-91.881,-36.893,179.593,5.313,149.046
C00619=1226.620,-91.632,-36.905,179.595,5.313,149.045
C00620=1226.614,-91.382,-36.915,179.597,5.313,149.045
C00621=1226.609,-91.133,-36.926,179.599,5.313,149.044
C00622=1226.604,-90.883,-36.936,179.602,5.313,149.043
C00623=1226.599,-90.633,-36.948,179.604,5.313,149.043
C00624=1226.593,-90.383,-36.959,179.607,5.313,149.042
C00625=1226.588,-90.134,-36.970,179.609,5.313,149.041
C00626=1226.583,-89.884,-36.980,179.611,5.314,149.041
C00627=1226.578,-89.635,-36.991,179.613,5.313,149.040
C00628=1226.573,-89.384,-37.002,179.616,5.314,149.039
C00629=1226.567,-89.135,-37.014,179.618,5.313,149.039
C00630=1226.562,-88.885,-37.024,179.621,5.314,149.038
C00631=1226.557,-88.635,-37.035,179.623,5.313,149.037
C00632=1226.552,-88.386,-37.046,179.625,5.314,149.036
C00633=1226.547,-88.136,-37.057,179.627,5.314,149.036
C00634=1226.541,-87.886,-37.069,179.630,5.314,149.035
C00635=1226.536,-87.636,-37.079,179.632,5.314,149.034
C00636=1226.531,-87.387,-37.090,179.635,5.314,149.034
C00637=1226.526,-87.137,-37.101,179.637,5.314,149.033
C00638=1226.520,-86.887,-37.112,179.640,5.314,149.032
C00639=1226.515,-86.638,-37.123,179.642,5.314,149.031
C00640=1226.510,-86.388,-37.134,179.644,5.314,149.031
C00641=1226.505,-86.138,-37.145,179.647,5.314,149.030
C00642=1226.499,-85.889,-37.157,179.649,5.314,149.029
C00643=1226.494,-85.639,-37.167,179.651,5.314,149.029
C00644=1226.490,-85.389,-37.179,179.654,5.314,149.028
C00645=1226.484,-85.140,-37.190,179.656,5.314,149.027
C00646=1226.479,-84.890,-37.201,179.658,5.315,149.027
C00647=1226.474,-84.640,-37.212,179.660,5.315,149.026
C00648=1226.469,-84.391,-37.223,179.663,5.315,149.025
C00649=1226.464,-84.141,-37.234,179.665,5.315,149.025
C00650=1226.458,-83.891,-37.245,179.668,5.315,149.024
C00651=1226.453,-83.642,-37.256,179.670,5.315,149.023
C00652=1226.448,-83.392,-37.267,179.673,5.315,149.022
C00653=1226.443,-83.142,-37.279,179.675,5.315,149.022
C00654=1226.438,-82.892,-37.290,179.677,5.315,149.021
C00655=1226.433,-82.643,-37.301,179.679,5.315,149.020
C00656=1226.427,-82.393,-37.312,179.682,5.315,149.020
C00657=1226.422,-82.143,-37.323,179.684,5.315,149.019
C00658=1226.417,-81.894,-37.334,179.687,5.315,149.018
C00659=1226.411,-81.643,-37.346,179.689,5.315,149.017
C00660=1226.406,-81.394,-37.357,179.692,5.316,149.017
C00661=1226.402,-81.144,-37.368,179.694,5.315,149.016
C00662=1226.396,-80.895,-37.380,179.696,5.316,149.015
C00663=1226.391,-80.645,-37.391,179.698,5.315,149.015
C00664=1226.386,-80.395,-37.402,179.701,5.316,149.014
C00665=1226.381,-80.145,-37.413,179.703,5.315,149.013
C00666=1226.375,-79.896,-37.424,179.706,5.316,149.012
C00667=1226.371,-79.647,-37.436,179.708,5.316,149.012
C00668=1226.365,-79.397,-37.448,179.711,5.316,149.011
C00669=1226.360,-79.146,-37.458,179.713,5.316,149.010
C00670=1226.354,-78.897,-37.470,179.715,5.316,149.010
C00671=1226.349,-78.648,-37.481,179.718,5.317,149.009
C00672=1226.345,-78.398,-37.492,179.720,5.317,149.008
C00673=1226.339,-78.148,-37.504,179.722,5.317,149.008
C00674=1226.334,-77.899,-37.515,179.724,5.317,149.007
C00675=1226.328,-77.649,-37.526,179.727,5.317,149.006
C00676=1226.324,-77.399,-37.537,179.729,5.317,149.006
C00677=1226.318,-77.149,-37.549,179.732,5.317,149.005
C00678=1226.314,-76.899,-37.561,179.734,5.317,149.004
C00679=1226.308,-76.650,-37.572,179.737,5.317,149.003
C00680=1226.303,-76.401,-37.583,179.739,5.317,149.003
C00681=1226.298,-76.151,-37.595,179.741,5.317,149.002
C00682=1226.293,-75.901,-37.607,179.743,5.317,149.001
C00683=1226.288,-75.651,-37.618,179.746,5.318,149.001
C00684=1226.282,-75.402,-37.629,179.748,5.317,149.000
C00685=1226.277,-75.152,-37.640,179.751,5.318,148.999
C00686=1226.272,-74.882,-37.653,179.753,5.317,148.999
C00687=1226.265,-74.611,-37.665,179.756,5.318,148.998
C00688=1226.260,-74.341,-37.678,179.759,5.318,148.997
C00689=1226.255,-74.070,-37.690,179.761,5.318,148.996
C00690=1226.249,-73.821,-37.701,179.764,5.318,148.995
C00691=1226.244,-73.571,-37.713,179.766,5.318,148.995
C00692=1226.238,-73.321,-37.725,179.768,5.318,148.994
C00693=1226.234,-73.071,-37.736,179.771,5.319,148.993
C00694=1226.228,-72.822,-37.748,179.773,5.318,148.993
C00695=1226.224,-72.572,-37.759,179.776,5.319,148.992
C00696=1226.218,-72.323,-37.771,179.778,5.318,148.991
C00697=1226.213,-72.073,-37.782,179.781,5.319,148.991
C00698=1226.207,-71.823,-37.794,179.783,5.318,148.990
C00699=1226.203,-71.573,-37.805,179.785,5.319,148.989
C00700=1226.198,-71.324,-37.818,179.787,5.319,148.988
C00701=1226.193,-71.075,-37.829,179.790,5.319,148.988
C00702=1226.187,-70.825,-37.841,179.792,5.319,148.987
C00703=1226.182,-70.575,-37.853,179.795,5.319,148.986
C00704=1226.177,-70.326,-37.864,179.797,5.319,148.986
C00705=1226.171,-70.076,-37.876,179.800,5.319,148.985
C00706=1226.167,-69.826,-37.887,179.802,5.320,148.984
C00707=1226.161,-69.576,-37.899,179.804,5.319,148.983
C00708=1226.157,-69.327,-37.910,179.807,5.320,148.983
C00709=1226.151,-69.077,-37.922,179.809,5.320,148.982
C00710=1226.146,-68.827,-37.934,179.811,5.320,148.982
C00711=1226.141,-68.577,-37.945,179.813,5.320,148.981
C00712=1226.136,-68.328,-37.958,179.816,5.320,148.980
C00713=1226.130,-68.079,-37.969,179.818,5.320,148.979
C00714=1226.125,-67.829,-37.981,179.821,5.321,148.979
C00715=1226.120,-67.579,-37.993,179.823,5.320,148.978
C00716=1226.115,-67.329,-38.004,179.826,5.321,148.977
C00717=1226.110,-67.079,-38.016,179.828,5.320,148.977
C00718=1226.104,-66.830,-38.028,179.830,5.321,148.976
C00719=1226.100,-66.581,-38.040,179.833,5.321,148.975
C00720=1226.094,-66.331,-38.051,179.835,5.321,148.974
C00721=1226.089,-66.081,-38.063,179.838,5.321,148.974
C00722=1226.084,-65.831,-38.075,179.840,5.321,148.973
C00723=1226.079,-65.581,-38.087,179.842,5.322,148.972
C00724=1226.074,-65.332,-38.099,179.845,5.321,148.972
C00725=1226.069,-65.082,-38.110,179.847,5.322,148.971
C00726=1226.063,-64.833,-38.122,179.849,5.321,148.970
C00727=1226.057,-64.583,-38.134,179.852,5.322,148.970
C00728=1226.053,-64.333,-38.145,179.855,5.322,148.969
C00729=1226.048,-64.084,-38.158,179.857,5.322,148.968
C00730=1226.042,-63.834,-38.170,179.859,5.322,148.967
C00731=1226.037,-63.584,-38.181,179.861,5.322,148.967
C00732=1226.032,-63.335,-38.193,179.864,5.323,148.966
C00733=1226.027,-63.085,-38.205,179.866,5.322,148.965
C00734=1226.022,-62.835,-38.217,179.869,5.323,148.965
C00735=1226.017,-62.586,-38.229,179.871,5.322,148.964
C00736=1226.012,-62.336,-38.241,179.874,5.323,148.963
C00737=1226.006,-62.086,-38.253,179.876,5.322,148.962
C00738=1226.001,-61.836,-38.265,179.878,5.323,148.962
C00739=1225.997,-61.587,-38.277,179.881,5.323,148.961
C00740=1225.991,-61.337,-38.289,179.883,5.323,148.960
C00741=1225.986,-61.088,-38.301,179.886,5.324,148.960
C00742=1225.981,-60.838,-38.313,179.888,5.323,148.959
C00743=1225.976,-60.589,-38.325,179.891,5.324,148.958
C00744=1225.970,-60.339,-38.336,179.893,5.323,148.958
C00745=1225.965,-60.089,-38.349,179.895,5.324,148.957
C00746=1225.960,-59.839,-38.361,179.898,5.324,148.956
C00747=1225.955,-59.590,-38.372,179.900,5.324,148.955
C00748=1225.950,-59.340,-38.385,179.903,5.324,148.955
C00749=1225.945,-59.091,-38.397,179.905,5.324,148.954
C00750=1225.939,-58.841,-38.409,179.908,5.325,148.953
C00751=1225.934,-58.591,-38.421,179.910,5.324,148.953
C00752=1225.929,-58.342,-38.433,179.912,5.325,148.952
C00753=1225.925,-58.092,-38.445,179.914,5.324,148.951
C00754=1225.919,-57.842,-38.457,179.917,5.325,148.950
C00755=1225.914,-57.592,-38.470,179.920,5.325,148.950
C00756=1225.909,-57.342,-38.482,179.922,5.325,148.949
C00757=1225.903,-57.093,-38.494,179.924,5.325,148.948
C00758=1225.899,-56.844,-38.506,179.927,5.325,148.948
C00759=1225.894,-56.594,-38.518,179.929,5.326,148.947
C00760=1225.888,-56.344,-38.530,179.931,5.325,148.946
C00761=1225.883,-56.094,-38.542,179.934,5.326,148.946
C00762=1225.878,-55.845,-38.555,179.937,5.326,148.945
C00763=1225.872,-55.595,-38.567,179.939,5.326,148.944
C00764=1225.867,-55.346,-38.579,179.941,5.326,148.943
C00765=1225.863,-55.096,-38.590,179.943,5.326,148.943
C00766=1225.858,-54.847,-38.603,179.946,5.326,148.942
C00767=1225.853,-54.596,-38.615,179.948,5.326,148.941
C00768=1225.848,-54.347,-38.628,179.951,5.327,148.941
C00769=1225.842,-54.097,-38.640,179.954,5.327,148.940
C00770=1225.837,-53.848,-38.652,179.956,5.327,148.939
C00771=1225.832,-53.598,-38.664,179.958,5.327,148.938
C00772=1225.827,-53.348,-38.677,179.960,5.327,148.938
C00773=1225.821,-53.099,-38.690,179.963,5.327,148.937
C00774=1225.816,-52.849,-38.701,179.966,5.328,148.936
C00775=1225.812,-52.600,-38.713,179.968,5.327,148.936
C00776=1225.807,-52.349,-38.726,179.970,5.328,148.935
C00777=1225.802,-52.100,-38.738,179.973,5.328,148.934
C00778=1225.796,-51.850,-38.750,179.975,5.328,148.934
C00779=1225.791,-51.601,-38.763,179.977,5.328,148.933
C00780=1225.786,-51.352,-38.775,179.980,5.328,148.932
C00781=1225.781,-51.102,-38.787,179.983,5.329,148.931
C00782=1225.775,-50.852,-38.800,179.985,5.328,148.931
C00783=1225.771,-50.602,-38.813,179.987,5.329,148.930
C00784=1225.765,-50.352,-38.825,179.989,5.329,148.929
C00785=1225.760,-50.103,-38.837,179.992,5.329,148.929
C00786=1225.755,-49.853,-38.849,179.995,5.330,148.928
C00787=1225.750,-49.604,-38.862,179.997,5.329,148.927
C00788=1225.745,-49.354,-38.874,180.000,5.330,148.927
C00789=1225.740,-49.104,-38.887,-179.998,5.329,148.926
C00790=1225.734,-48.835,-38.900,-179.996,5.330,148.925
C00791=1225.728,-48.565,-38.914,-179.992,5.330,148.924
C00792=1225.723,-48.295,-38.927,-179.990,5.330,148.923
C00793=1225.718,-48.025,-38.940,-179.988,5.330,148.923
C00794=1225.712,-47.776,-38.953,-179.985,5.331,148.922
C00795=1225.708,-47.525,-38.965,-179.983,5.330,148.921
C00796=1225.702,-47.276,-38.978,-179.980,5.331,148.921
C00797=1225.697,-47.027,-38.991,-179.978,5.331,148.920
C00798=1225.692,-46.777,-39.003,-179.976,5.331,148.919
C00799=1225.686,-46.527,-39.016,-179.973,5.331,148.919
C00800=1225.681,-46.278,-39.028,-179.971,5.331,148.918
C00801=1225.676,-46.028,-39.041,-179.968,5.331,148.917
C00802=1225.671,-45.779,-39.054,-179.965,5.332,148.916
C00803=1225.666,-45.529,-39.066,-179.963,5.332,148.916
C00804=1225.661,-45.279,-39.078,-179.961,5.332,148.915
C00805=1225.656,-45.029,-39.091,-179.959,5.332,148.914
C00806=1225.651,-44.780,-39.104,-179.956,5.332,148.914
C00807=1225.646,-44.531,-39.116,-179.953,5.333,148.913
C00808=1225.641,-44.281,-39.128,-179.951,5.332,148.912
C00809=1225.635,-44.031,-39.141,-179.949,5.333,148.912
C00810=1225.630,-43.781,-39.154,-179.947,5.333,148.911
C00811=1225.625,-43.532,-39.167,-179.944,5.333,148.910
C00812=1225.620,-43.282,-39.180,-179.941,5.334,148.909
C00813=1225.615,-43.033,-39.192,-179.939,5.333,148.909
C00814=1225.610,-42.782,-39.205,-179.936,5.334,148.908
C00815=1225.605,-42.533,-39.217,-179.934,5.333,148.907
C00816=1225.600,-42.284,-39.230,-179.932,5.334,148.907
C00817=1225.594,-42.034,-39.243,-179.929,5.334,148.906
C00818=1225.589,-41.784,-39.256,-179.927,5.334,148.905
C00819=1225.584,-41.535,-39.269,-179.924,5.335,148.905
C00820=1225.579,-41.286,-39.281,-179.922,5.334,148.904
C00821=1225.575,-41.036,-39.294,-179.920,5.335,148.903
C00822=1225.569,-40.786,-39.307,-179.917,5.335,148.902
C00823=1225.564,-40.537,-39.320,-179.915,5.335,148.902
C00824=1225.558,-40.287,-39.332,-179.912,5.335,148.901
C00825=1225.554,-40.037,-39.345,-179.910,5.335,148.900
C00826=1225.548,-39.787,-39.357,-179.907,5.336,148.900
C00827=1225.543,-39.538,-39.370,-179.905,5.336,148.899
C00828=1225.538,-39.288,-39.383,-179.903,5.336,148.898
C00829=1225.533,-39.038,-39.396,-179.900,5.336,148.898
C00830=1225.528,-38.789,-39.409,-179.897,5.337,148.897
C00831=1225.523,-38.539,-39.422,-179.895,5.336,148.896
C00832=1225.518,-38.290,-39.434,-179.893,5.337,148.895
C00833=1225.512,-38.040,-39.447,-179.890,5.337,148.895
C00834=1225.508,-37.790,-39.460,-179.888,5.337,148.894
C00835=1225.503,-37.541,-39.473,-179.885,5.337,148.893
C00836=1225.498,-37.291,-39.486,-179.883,5.337,148.893
C00837=1225.492,-37.042,-39.499,-179.880,5.338,148.892
C00838=1225.487,-36.792,-39.512,-179.878,5.338,148.891
C00839=1225.482,-36.542,-39.524,-179.876,5.338,148.891
C00840=1225.476,-36.293,-39.538,-179.873,5.338,148.890
C00841=1225.472,-36.043,-39.551,-179.871,5.338,148.889
C00842=1225.467,-35.793,-39.563,-179.868,5.338,148.888
C00843=1225.462,-35.544,-39.577,-179.866,5.339,148.888
C00844=1225.456,-35.294,-39.590,-179.863,5.339,148.887
C00845=1225.451,-35.045,-39.603,-179.861,5.339,148.886
C00846=1225.447,-34.795,-39.616,-179.858,5.340,148.886
C00847=1225.441,-34.546,-39.629,-179.856,5.339,148.885
C00848=1225.436,-34.296,-39.641,-179.853,5.340,148.884
C00849=1225.431,-34.046,-39.654,-179.851,5.339,148.884
C00850=1225.425,-33.797,-39.668,-179.849,5.340,148.883
C00851=1225.420,-33.547,-39.680,-179.846,5.340,148.882
C00852=1225.416,-33.298,-39.694,-179.844,5.340,148.881
C00853=1225.410,-33.048,-39.707,-179.841,5.341,148.881
C00854=1225.406,-32.798,-39.720,-179.839,5.341,148.880
C00855=1225.401,-32.549,-39.733,-179.837,5.341,148.879
C00856=1225.395,-32.299,-39.746,-179.834,5.341,148.879
C00857=1225.390,-32.049,-39.759,-179.831,5.342,148.878
C00858=1225.385,-31.800,-39.771,-179.829,5.342,148.877
C00859=1225.380,-31.550,-39.786,-179.826,5.342,148.877
C00860=1225.375,-31.301,-39.798,-179.824,5.342,148.876
C00861=1225.369,-31.051,-39.811,-179.822,5.342,148.875
C00862=1225.365,-30.801,-39.824,-179.819,5.343,148.874
C00863=1225.360,-30.553,-39.838,-179.816,5.342,148.874
C00864=1225.355,-30.302,-39.851,-179.814,5.342,148.873
C00865=1225.349,-30.053,-39.864,-179.811,5.343,148.872
C00866=1225.344,-29.803,-39.877,-179.809,5.343,148.871
C00867=1225.339,-29.553,-39.890,-179.806,5.343,148.871
C00868=1225.334,-29.305,-39.903,-179.804,5.344,148.870
C00869=1225.329,-29.054,-39.917,-179.802,5.343,148.869
C00870=1225.324,-28.805,-39.930,-179.799,5.344,148.869
C00871=1225.319,-28.555,-39.944,-179.796,5.344,148.868
C00872=1225.314,-28.306,-39.956,-179.794,5.344,148.867
C00873=1225.309,-28.056,-39.970,-179.792,5.345,148.867
C00874=1225.303,-27.806,-39.983,-179.790,5.344,148.866
C00875=1225.299,-27.557,-39.996,-179.787,5.345,148.865
C00876=1225.293,-27.307,-40.009,-179.784,5.345,148.864
C00877=1225.289,-27.057,-40.022,-179.782,5.345,148.864
C00878=1225.283,-26.808,-40.036,-179.779,5.345,148.863
C00879=1225.279,-26.558,-40.049,-179.777,5.346,148.862
C00880=1225.273,-26.308,-40.062,-179.775,5.346,148.862
C00881=1225.269,-26.059,-40.076,-179.772,5.346,148.861
C00882=1225.263,-25.809,-40.089,-179.769,5.347,148.860
C00883=1225.258,-25.559,-40.102,-179.767,5.346,148.860
C00884=1225.253,-25.310,-40.116,-179.765,5.347,148.859
C00885=1225.248,-25.060,-40.129,-179.762,5.347,148.858
C00886=1225.243,-24.811,-40.143,-179.760,5.347,148.858
C00887=1225.238,-24.561,-40.156,-179.757,5.347,148.857
C00888=1225.232,-24.312,-40.169,-179.755,5.348,148.856
C00889=1225.228,-24.062,-40.183,-179.753,5.348,148.855
C00890=1225.222,-23.813,-40.196,-179.750,5.348,148.855
C00891=1225.218,-23.563,-40.210,-179.747,5.349,148.854
C00892=1225.212,-23.314,-40.223,-179.745,5.348,148.853
C00893=1225.207,-23.064,-40.237,-179.742,5.349,148.853
C00894=1225.202,-22.795,-40.251,-179.740,5.349,148.852
C00895=1225.196,-22.526,-40.266,-179.737,5.350,148.851
C00896=1225.191,-22.256,-40.281,-179.735,5.350,148.851
C00897=1225.186,-21.986,-40.294,-179.732,5.350,148.850
C00898=1225.180,-21.737,-40.308,-179.729,5.350,148.849
C00899=1225.175,-21.487,-40.322,-179.727,5.351,148.848
C00900=1225.170,-21.238,-40.335,-179.724,5.350,148.848
C00901=1225.165,-20.988,-40.349,-179.722,5.351,148.847
C00902=1225.160,-20.739,-40.362,-179.719,5.351,148.846
C00903=1225.155,-20.489,-40.376,-179.717,5.351,148.845
C00904=1225.150,-20.239,-40.390,-179.714,5.352,148.845
C00905=1225.145,-19.990,-40.402,-179.712,5.352,148.844
C00906=1225.140,-19.740,-40.417,-179.710,5.352,148.843
C00907=1225.134,-19.491,-40.431,-179.707,5.352,148.843
C00908=1225.130,-19.241,-40.444,-179.704,5.353,148.842
C00909=1225.124,-18.992,-40.457,-179.702,5.352,148.841
C00910=1225.119,-18.742,-40.471,-179.700,5.353,148.841
C00911=1225.115,-18.493,-40.485,-179.697,5.353,148.840
C00912=1225.109,-18.243,-40.498,-179.695,5.353,148.839
C00913=1225.104,-17.993,-40.512,-179.692,5.354,148.838
C00914=1225.099,-17.744,-40.525,-179.690,5.354,148.838
C00915=1225.094,-17.494,-40.539,-179.688,5.354,148.837
C00916=1225.089,-17.244,-40.553,-179.685,5.354,148.836
C00917=1225.084,-16.995,-40.566,-179.682,5.355,148.836
C00918=1225.079,-16.745,-40.580,-179.680,5.355,148.835
C00919=1225.073,-16.496,-40.594,-179.677,5.355,148.834
C00920=1225.069,-16.246,-40.607,-179.675,5.356,148.834
C00921=1225.064,-15.997,-40.621,-179.672,5.356,148.833
C00922=1225.058,-15.748,-40.635,-179.670,5.356,148.832
C00923=1225.053,-15.498,-40.648,-179.667,5.356,148.832
C00924=1225.049,-15.248,-40.663,-179.665,5.357,148.831
C00925=1225.043,-14.999,-40.676,-179.663,5.356,148.830
C00926=1225.038,-14.749,-40.690,-179.660,5.357,148.829
C00927=1225.033,-14.499,-40.704,-179.657,5.358,148.829
C00928=1225.028,-14.250,-40.718,-179.655,5.357,148.828
C00929=1225.023,-14.000,-40.732,-179.653,5.358,148.827
C00930=1225.018,-13.750,-40.745,-179.650,5.358,148.827
C00931=1225.013,-13.501,-40.759,-179.648,5.358,148.826
C00932=1225.008,-13.252,-40.773,-179.645,5.358,148.825
C00933=1225.003,-13.002,-40.787,-179.643,5.359,148.825
C00934=1224.997,-12.752,-40.800,-179.640,5.359,148.824
C00935=1224.993,-12.503,-40.814,-179.638,5.359,148.823
C00936=1224.988,-12.253,-40.828,-179.635,5.360,148.823
C00937=1224.982,-12.004,-40.842,-179.633,5.360,148.822
C00938=1224.977,-11.754,-40.856,-179.630,5.360,148.821
C00939=1224.972,-11.504,-40.870,-179.628,5.360,148.820
C00940=1224.967,-11.256,-40.884,-179.625,5.361,148.820
C00941=1224.962,-11.006,-40.898,-179.623,5.361,148.819
C00942=1224.957,-10.756,-40.912,-179.620,5.361,148.818
C00943=1224.952,-10.506,-40.925,-179.618,5.362,148.818
C00944=1224.947,-10.257,-40.940,-179.615,5.362,148.817
C00945=1224.942,-10.007,-40.954,-179.613,5.362,148.816
C00946=1224.937,-9.758,-40.968,-179.610,5.362,148.816
C00947=1224.932,-9.509,-40.981,-179.608,5.363,148.815
C00948=1224.927,-9.259,-40.996,-179.606,5.363,148.814
C00949=1224.922,-9.009,-41.010,-179.603,5.363,148.814
C00950=1224.917,-8.759,-41.024,-179.601,5.364,148.813
C00951=1224.911,-8.510,-41.037,-179.598,5.364,148.812
C00952=1224.906,-8.260,-41.052,-179.596,5.364,148.812
C00953=1224.902,-8.011,-41.065,-179.593,5.365,148.811
C00954=1224.897,-7.761,-41.080,-179.591,5.365,148.810
C00955=1224.892,-7.512,-41.094,-179.589,5.365,148.810
C00956=1224.887,-7.262,-41.108,-179.586,5.365,148.809
C00957=1224.882,-7.013,-41.122,-179.583,5.366,148.808
C00958=1224.877,-6.763,-41.136,-179.581,5.366,148.808
C00959=1224.871,-6.514,-41.150,-179.579,5.366,148.807
C00960=1224.866,-6.264,-41.165,-179.576,5.367,148.806
C00961=1224.861,-6.015,-41.179,-179.573,5.367,148.805
C00962=1224.856,-5.765,-41.193,-179.571,5.368,148.805
C00963=1224.851,-5.516,-41.206,-179.569,5.367,148.804
C00964=1224.846,-5.266,-41.221,-179.566,5.368,148.803
C00965=1224.842,-5.017,-41.235,-179.563,5.368,148.803
C00966=1224.837,-4.767,-41.249,-179.561,5.368,148.802
C00967=1224.832,-4.517,-41.264,-179.559,5.369,148.801
C00968=1224.826,-4.268,-41.278,-179.556,5.369,148.801
C00969=1224.821,-4.019,-41.292,-179.553,5.370,148.800
C00970=1224.816,-3.769,-41.306,-179.551,5.369,148.799
C00971=1224.811,-3.519,-41.320,-179.548,5.370,148.799
C00972=1224.806,-3.269,-41.335,-179.546,5.370,148.798
C00973=1224.801,-3.020,-41.349,-179.543,5.371,148.797
C00974=1224.796,-2.771,-41.363,-179.541,5.371,148.796
C00975=1224.791,-2.521,-41.377,-179.538,5.371,148.796
C00976=1224.786,-2.271,-41.391,-179.536,5.372,148.795
C00977=1224.781,-2.022,-41.406,-179.533,5.372,148.794
C00978=1224.776,-1.772,-41.420,-179.531,5.372,148.794
C00979=1224.770,-1.523,-41.434,-179.528,5.372,148.793
C00980=1224.765,-1.273,-41.448,-179.526,5.373,148.792
C00981=1224.760,-1.023,-41.462,-179.524,5.373,148.792
C00982=1224.756,-0.774,-41.477,-179.521,5.373,148.791
C00983=1224.751,-0.525,-41.492,-179.518,5.374,148.790
C00984=1224.746,-0.275,-41.506,-179.516,5.374,148.790
C00985=1224.740,-0.026,-41.520,-179.514,5.374,148.789
C00986=1224.735,0.224,-41.534,-179.511,5.374,148.788
C00987=1224.730,0.474,-41.549,-179.508,5.375,148.788
C00988=1224.725,0.723,-41.564,-179.506,5.375,148.787
C00989=1224.720,0.973,-41.578,-179.504,5.375,148.786
C00990=1224.715,1.222,-41.593,-179.501,5.376,148.785
C00991=1224.710,1.472,-41.607,-179.498,5.376,148.785
C00992=1224.705,1.722,-41.621,-179.496,5.377,148.784
C00993=1224.700,1.971,-41.635,-179.494,5.376,148.783
C00994=1224.695,2.220,-41.650,-179.491,5.377,148.783
C00995=1224.690,2.470,-41.664,-179.488,5.378,148.782
C00996=1224.685,2.719,-41.679,-179.486,5.378,148.781
C00997=1224.679,2.969,-41.693,-179.484,5.378,148.781
C00998=1224.674,3.238,-41.709,-179.481,5.378,148.780
C00999=1224.669,3.507,-41.725,-179.478,5.379,148.779
C01000=1224.664,3.776,-41.741,-179.476,5.379,148.779
C01001=1224.659,4.045,-41.756,-179.472,5.379,148.778
C01002=1224.653,4.295,-41.771,-179.470,5.380,148.777
C01003=1224.648,4.544,-41.785,-179.468,5.381,148.777
C01004=1224.643,4.793,-41.799,-179.466,5.381,148.776
C01005=1224.638,5.042,-41.814,-179.463,5.381,148.775
C01006=1224.633,5.292,-41.829,-179.460,5.382,148.774
C01007=1224.628,5.542,-41.843,-179.458,5.382,148.774
C01008=1224.623,5.791,-41.858,-179.456,5.382,148.773
C01009=1224.618,6.041,-41.873,-179.453,5.382,148.772
C01010=1224.613,6.291,-41.887,-179.450,5.383,148.772
C01011=1224.608,6.540,-41.902,-179.448,5.383,148.771
C01012=1224.603,6.789,-41.916,-179.445,5.384,148.770
C01013=1224.598,7.039,-41.931,-179.443,5.384,148.770
C01014=1224.593,7.288,-41.946,-179.440,5.384,148.769
C01015=1224.588,7.538,-41.960,-179.438,5.385,148.768
C01016=1224.583,7.787,-41.975,-179.435,5.385,148.768
C01017=1224.578,8.037,-41.990,-179.433,5.385,148.767
C01018=1224.573,8.287,-42.005,-179.430,5.386,148.766
C01019=1224.568,8.536,-42.020,-179.428,5.386,148.766
C01020=1224.563,8.786,-42.034,-179.425,5.387,148.765
C01021=1224.558,9.035,-42.049,-179.423,5.386,148.764
C01022=1224.553,9.285,-42.064,-179.420,5.387,148.763
C01023=1224.548,9.534,-42.079,-179.417,5.387,148.763
C01024=1224.543,9.784,-42.093,-179.415,5.388,148.762
C01025=1224.537,10.034,-42.108,-179.412,5.388,148.761
C01026=1224.533,10.283,-42.123,-179.410,5.388,148.761
C01027=1224.528,10.533,-42.137,-179.407,5.389,148.760
C01028=1224.523,10.782,-42.152,-179.405,5.389,148.759
C01029=1224.517,11.032,-42.167,-179.402,5.390,148.759
C01030=1224.513,11.281,-42.182,-179.400,5.390,148.758
C01031=1224.508,11.530,-42.196,-179.397,5.390,148.757
C01032=1224.502,11.780,-42.212,-179.395,5.391,148.757
C01033=1224.497,12.030,-42.226,-179.393,5.391,148.756
C01034=1224.493,12.279,-42.241,-179.390,5.392,148.755
C01035=1224.487,12.529,-42.256,-179.387,5.392,148.755
C01036=1224.482,12.778,-42.271,-179.385,5.392,148.754
C01037=1224.478,13.027,-42.286,-179.383,5.393,148.753
C01038=1224.472,13.277,-42.301,-179.380,5.393,148.753
C01039=1224.468,13.526,-42.316,-179.377,5.394,148.752
C01040=1224.463,13.776,-42.330,-179.375,5.394,148.751
C01041=1224.457,14.025,-42.346,-179.373,5.394,148.751
C01042=1224.453,14.274,-42.361,-179.370,5.395,148.750
C01043=1224.448,14.524,-42.375,-179.367,5.395,148.749
C01044=1224.442,14.773,-42.391,-179.365,5.396,148.749
C01045=1224.438,15.024,-42.405,-179.362,5.396,148.748
C01046=1224.432,15.273,-42.421,-179.360,5.396,148.747
C01047=1224.428,15.522,-42.436,-179.357,5.396,148.747
C01048=1224.423,15.772,-42.450,-179.355,5.397,148.746
C01049=1224.417,16.021,-42.466,-179.352,5.397,148.745
C01050=1224.413,16.270,-42.481,-179.349,5.398,148.745
C01051=1224.407,16.520,-42.495,-179.347,5.398,148.744
C01052=1224.402,16.770,-42.510,-179.345,5.398,148.743
C01053=1224.397,17.019,-42.526,-179.342,5.399,148.742
C01054=1224.392,17.269,-42.540,-179.340,5.400,148.742
C01055=1224.387,17.518,-42.555,-179.337,5.400,148.741
C01056=1224.383,17.768,-42.571,-179.335,5.400,148.741
C01057=1224.378,18.018,-42.586,-179.332,5.400,148.740
C01058=1224.372,18.267,-42.601,-179.330,5.401,148.739
C01059=1224.368,18.516,-42.616,-179.327,5.402,148.739
C01060=1224.362,18.765,-42.632,-179.324,5.402,148.738
C01061=1224.357,19.015,-42.646,-179.322,5.403,148.737
C01062=1224.352,19.265,-42.662,-179.320,5.402,148.737
C01063=1224.348,19.514,-42.677,-179.317,5.403,148.736
C01064=1224.343,19.764,-42.693,-179.314,5.403,148.735
C01065=1224.338,20.013,-42.707,-179.312,5.404,148.735
C01066=1224.332,20.263,-42.722,-179.309,5.404,148.734
C01067=1224.328,20.512,-42.737,-179.307,5.404,148.733
C01068=1224.322,20.761,-42.753,-179.304,5.405,148.732
C01069=1224.317,21.010,-42.768,-179.302,5.405,148.732
C01070=1224.312,21.261,-42.783,-179.299,5.406,148.731
C01071=1224.308,21.510,-42.798,-179.297,5.407,148.731
C01072=1224.302,21.760,-42.814,-179.294,5.407,148.730
C01073=1224.298,22.009,-42.829,-179.292,5.407,148.729
C01074=1224.292,22.258,-42.844,-179.290,5.408,148.729
C01075=1224.288,22.508,-42.860,-179.287,5.408,148.728
C01076=1224.283,22.757,-42.875,-179.284,5.409,148.727
C01077=1224.277,23.007,-42.890,-179.282,5.409,148.727
C01078=1224.273,23.256,-42.905,-179.279,5.410,148.726
C01079=1224.267,23.506,-42.921,-179.277,5.409,148.725
C01080=1224.263,23.756,-42.936,-179.274,5.410,148.725
C01081=1224.258,24.005,-42.952,-179.272,5.411,148.724
C01082=1224.252,24.254,-42.967,-179.269,5.411,148.723
C01083=1224.248,24.504,-42.982,-179.266,5.412,148.722
C01084=1224.242,24.753,-42.998,-179.264,5.412,148.722
C01085=1224.238,25.003,-43.013,-179.262,5.412,148.721
C01086=1224.233,25.252,-43.029,-179.260,5.413,148.721
C01087=1224.227,25.502,-43.044,-179.257,5.413,148.720
C01088=1224.223,25.751,-43.059,-179.254,5.414,148.719
C01089=1224.218,26.001,-43.075,-179.252,5.414,148.719
C01090=1224.213,26.250,-43.091,-179.249,5.415,148.718
C01091=1224.208,26.499,-43.106,-179.246,5.415,148.717
C01092=1224.203,26.749,-43.122,-179.244,5.415,148.717
C01093=1224.199,26.998,-43.137,-179.242,5.416,148.716
C01094=1224.193,27.248,-43.152,-179.239,5.416,148.715
C01095=1224.188,27.497,-43.168,-179.236,5.417,148.715
C01096=1224.182,27.747,-43.184,-179.234,5.417,148.714
C01097=1224.178,27.996,-43.199,-179.231,5.418,148.713
C01098=1224.173,28.246,-43.215,-179.228,5.418,148.713
C01099=1224.168,28.495,-43.230,-179.226,5.418,148.712
C01100=1224.163,28.744,-43.245,-179.224,5.419,148.711
C01101=1224.158,28.994,-43.261,-179.222,5.420,148.711
C01102=1224.153,29.263,-43.278,-179.218,5.420,148.710
C01103=1224.147,29.532,-43.294,-179.216,5.420,148.709
C01104=1224.142,29.800,-43.311,-179.213,5.421,148.708
C01105=1224.136,30.069,-43.328,-179.210,5.421,148.708
C01106=1224.132,30.319,-43.344,-179.208,5.422,148.707
C01107=1224.126,30.568,-43.359,-179.205,5.423,148.706
C01108=1224.122,30.817,-43.374,-179.203,5.423,148.706
C01109=1224.116,31.066,-43.391,-179.200,5.424,148.705
C01110=1224.112,31.316,-43.407,-179.197,5.424,148.704
C01111=1224.106,31.566,-43.422,-179.196,5.424,148.704
C01112=1224.102,31.815,-43.437,-179.193,5.425,148.703
C01113=1224.097,32.065,-43.453,-179.190,5.425,148.703
C01114=1224.091,32.314,-43.469,-179.188,5.426,148.702
C01115=1224.086,32.563,-43.485,-179.185,5.426,148.701
C01116=1224.082,32.813,-43.500,-179.182,5.427,148.701
C01117=1224.077,33.062,-43.516,-179.180,5.428,148.700
C01118=1224.072,33.312,-43.532,-179.177,5.428,148.699
C01119=1224.067,33.562,-43.548,-179.175,5.428,148.699
C01120=1224.062,33.810,-43.564,-179.172,5.428,148.698
C01121=1224.058,34.060,-43.579,-179.170,5.429,148.697
C01122=1224.052,34.310,-43.595,-179.168,5.430,148.697
C01123=1224.047,34.559,-43.610,-179.165,5.430,148.696
C01124=1224.042,34.808,-43.627,-179.162,5.431,148.695
C01125=1224.037,35.058,-43.643,-179.160,5.432,148.695
C01126=1224.032,35.307,-43.658,-179.157,5.432,148.694
C01127=1224.027,35.557,-43.674,-179.154,5.433,148.693
C01128=1224.022,35.806,-43.690,-179.152,5.432,148.693
C01129=1224.018,36.056,-43.706,-179.150,5.433,148.692
C01130=1224.012,36.305,-43.722,-179.147,5.433,148.691
C01131=1224.007,36.554,-43.738,-179.144,5.434,148.691
C01132=1224.002,36.804,-43.754,-179.142,5.435,148.690
C01133=1223.997,37.054,-43.769,-179.140,5.435,148.690
C01134=1223.993,37.303,-43.786,-179.137,5.436,148.689
C01135=1223.987,37.553,-43.802,-179.134,5.437,148.688
C01136=1223.982,37.802,-43.817,-179.132,5.437,148.687
C01137=1223.978,38.051,-43.833,-179.130,5.437,148.687
C01138=1223.973,38.301,-43.849,-179.127,5.437,148.686
C01139=1223.968,38.551,-43.865,-179.124,5.438,148.685
C01140=1223.963,38.799,-43.881,-179.122,5.439,148.685
C01141=1223.957,39.049,-43.897,-179.120,5.439,148.684
C01142=1223.953,39.298,-43.913,-179.117,5.440,148.684
C01143=1223.948,39.548,-43.929,-179.114,5.441,148.683
C01144=1223.943,39.797,-43.946,-179.112,5.441,148.682
C01145=1223.938,40.047,-43.961,-179.109,5.442,148.682
C01146=1223.933,40.297,-43.977,-179.106,5.442,148.681
C01147=1223.928,40.545,-43.993,-179.104,5.443,148.680
C01148=1223.923,40.796,-44.009,-179.102,5.443,148.680
C01149=1223.918,41.044,-44.026,-179.099,5.443,148.679
C01150=1223.913,41.294,-44.042,-179.097,5.444,148.678
C01151=1223.908,41.543,-44.058,-179.094,5.445,148.678
C01152=1223.903,41.793,-44.074,-179.092,5.445,148.677
C01153=1223.898,42.042,-44.090,-179.089,5.446,148.676
C01154=1223.893,42.292,-44.106,-179.086,5.446,148.676
C01155=1223.888,42.541,-44.122,-179.084,5.447,148.675
C01156=1223.883,42.790,-44.138,-179.081,5.447,148.674
C01157=1223.879,43.040,-44.155,-179.078,5.448,148.674
C01158=1223.873,43.289,-44.170,-179.076,5.448,148.673
C01159=1223.869,43.539,-44.187,-179.074,5.449,148.673
C01160=1223.863,43.788,-44.203,-179.072,5.449,148.672
C01161=1223.859,44.038,-44.219,-179.069,5.450,148.671
C01162=1223.854,44.286,-44.236,-179.066,5.450,148.671
C01163=1223.849,44.537,-44.252,-179.064,5.451,148.670
C01164=1223.844,44.785,-44.268,-179.061,5.451,148.669
C01165=1223.839,45.035,-44.284,-179.058,5.452,148.669
C01166=1223.834,45.284,-44.300,-179.056,5.452,148.668
C01167=1223.829,45.534,-44.317,-179.054,5.453,148.668
C01168=1223.824,45.784,-44.333,-179.051,5.454,148.667
C01169=1223.819,46.033,-44.350,-179.048,5.454,148.666
C01170=1223.814,46.283,-44.366,-179.046,5.455,148.666
C01171=1223.809,46.532,-44.382,-179.043,5.456,148.665
C01172=1223.805,46.781,-44.399,-179.040,5.456,148.664
C01173=1223.799,47.031,-44.414,-179.038,5.457,148.663
C01174=1223.795,47.280,-44.431,-179.036,5.458,148.663
C01175=1223.790,47.529,-44.447,-179.033,5.458,148.662
C01176=1223.784,47.779,-44.464,-179.031,5.458,148.662
C01177=1223.780,48.029,-44.480,-179.028,5.459,148.661
C01178=1223.774,48.278,-44.497,-179.026,5.459,148.660
C01179=1223.770,48.527,-44.513,-179.023,5.460,148.660
C01180=1223.765,48.777,-44.529,-179.020,5.460,148.659
C01181=1223.760,49.026,-44.546,-179.018,5.461,148.659
C01182=1223.754,49.275,-44.562,-179.016,5.462,148.658
C01183=1223.750,49.525,-44.579,-179.013,5.462,148.657
C01184=1223.745,49.775,-44.595,-179.010,5.463,148.657
C01185=1223.740,50.023,-44.611,-179.008,5.463,148.656
C01186=1223.735,50.273,-44.628,-179.005,5.464,148.655
C01187=1223.730,50.522,-44.644,-179.002,5.464,148.655
C01188=1223.725,50.772,-44.661,-179.000,5.465,148.654
C01189=1223.720,51.022,-44.678,-178.998,5.466,148.653
C01190=1223.715,51.270,-44.694,-178.995,5.467,148.653
C01191=1223.711,51.520,-44.711,-178.992,5.467,148.652
C01192=1223.706,51.770,-44.728,-178.990,5.468,148.651
C01193=1223.700,52.019,-44.743,-178.987,5.468,148.651
C01194=1223.696,52.269,-44.760,-178.984,5.469,148.650
C01195=1223.691,52.517,-44.776,-178.982,5.470,148.650
C01196=1223.685,52.767,-44.794,-178.980,5.470,148.649
C01197=1223.681,53.017,-44.810,-178.977,5.471,148.648
C01198=1223.676,53.265,-44.827,-178.974,5.471,148.648
C01199=1223.671,53.515,-44.843,-178.972,5.472,148.647
C01200=1223.666,53.765,-44.861,-178.970,5.472,148.646
C01201=1223.661,54.014,-44.876,-178.967,5.472,148.646
C01202=1223.656,54.264,-44.893,-178.965,5.473,148.645
C01203=1223.652,54.513,-44.909,-178.962,5.474,148.645
C01204=1223.646,54.762,-44.926,-178.960,5.474,148.644
C01205=1223.642,55.012,-44.943,-178.957,5.475,148.643
C01206=1223.637,55.280,-44.961,-178.954,5.475,148.643
C01207=1223.631,55.548,-44.979,-178.951,5.477,148.642
C01208=1223.625,55.817,-44.996,-178.949,5.477,148.641
C01209=1223.620,56.086,-45.015,-178.946,5.478,148.641
C01210=1223.615,56.335,-45.032,-178.943,5.479,148.640
C01211=1223.610,56.584,-45.048,-178.941,5.479,148.639
C01212=1223.605,56.834,-45.065,-178.938,5.480,148.639
C01213=1223.601,57.083,-45.082,-178.936,5.481,148.638
C01214=1223.596,57.332,-45.098,-178.933,5.481,148.637
C01215=1223.590,57.582,-45.116,-178.931,5.482,148.637
C01216=1223.586,57.831,-45.132,-178.928,5.482,148.636
C01217=1223.581,58.081,-45.150,-178.925,5.483,148.635
C01218=1223.576,58.330,-45.166,-178.923,5.483,148.635
C01219=1223.571,58.579,-45.183,-178.921,5.484,148.634
C01220=1223.566,58.829,-45.200,-178.918,5.485,148.634
C01221=1223.562,59.078,-45.217,-178.915,5.486,148.633
C01222=1223.556,59.327,-45.234,-178.913,5.486,148.632
C01223=1223.551,59.577,-45.251,-178.910,5.487,148.632
C01224=1223.547,59.826,-45.267,-178.907,5.487,148.631
C01225=1223.542,60.076,-45.285,-178.905,5.488,148.631
C01226=1223.537,60.325,-45.301,-178.903,5.489,148.630
C01227=1223.531,60.575,-45.318,-178.900,5.489,148.629
C01228=1223.527,60.824,-45.335,-178.897,5.490,148.629
C01229=1223.522,61.074,-45.352,-178.895,5.490,148.628
C01230=1223.517,61.322,-45.369,-178.893,5.491,148.627
C01231=1223.512,61.572,-45.386,-178.890,5.492,148.627
C01232=1223.507,61.821,-45.403,-178.887,5.493,148.626
C01233=1223.503,62.071,-45.420,-178.885,5.493,148.625
C01234=1223.497,62.320,-45.437,-178.882,5.494,148.625
C01235=1223.493,62.569,-45.453,-178.880,5.495,148.624
C01236=1223.488,62.818,-45.471,-178.877,5.495,148.624
C01237=1223.483,63.068,-45.488,-178.875,5.496,148.623
C01238=1223.478,63.318,-45.505,-178.872,5.496,148.622
C01239=1223.473,63.567,-45.522,-178.869,5.497,148.622
C01240=1223.468,63.816,-45.540,-178.867,5.498,148.621
C01241=1223.463,64.066,-45.557,-178.865,5.498,148.621
C01242=1223.458,64.315,-45.574,-178.862,5.499,148.620
C01243=1223.453,64.565,-45.591,-178.859,5.500,148.619
C01244=1223.449,64.814,-45.608,-178.857,5.500,148.619
C01245=1223.443,65.063,-45.625,-178.854,5.501,148.618
C01246=1223.439,65.312,-45.642,-178.852,5.502,148.618
C01247=1223.433,65.562,-45.659,-178.849,5.502,148.617
C01248=1223.429,65.811,-45.676,-178.847,5.503,148.616
C01249=1223.424,66.061,-45.694,-178.844,5.503,148.616
C01250=1223.419,66.310,-45.710,-178.841,5.504,148.615
C01251=1223.414,66.559,-45.728,-178.839,5.505,148.614
C01252=1223.409,66.808,-45.745,-178.837,5.505,148.614
C01253=1223.404,67.058,-45.762,-178.834,5.506,148.613
C01254=1223.399,67.307,-45.780,-178.831,5.507,148.612
C01255=1223.395,67.557,-45.797,-178.829,5.507,148.612
C01256=1223.390,67.806,-45.814,-178.827,5.508,148.611
C01257=1223.385,68.056,-45.832,-178.823,5.510,148.611
C01258=1223.380,68.305,-45.848,-178.821,5.510,148.610
C01259=1223.375,68.554,-45.866,-178.818,5.511,148.609
C01260=1223.369,68.803,-45.883,-178.816,5.512,148.609
C01261=1223.365,69.053,-45.900,-178.813,5.512,148.608
C01262=1223.360,69.302,-45.918,-178.811,5.513,148.608
C01263=1223.356,69.551,-45.935,-178.808,5.513,148.607
C01264=1223.351,69.801,-45.953,-178.805,5.514,148.606
C01265=1223.345,70.050,-45.970,-178.803,5.515,148.606
C01266=1223.341,70.299,-45.987,-178.801,5.515,148.605
C01267=1223.336,70.549,-46.005,-178.798,5.516,148.605
C01268=1223.331,70.798,-46.022,-178.795,5.517,148.604
C01269=1223.326,71.048,-46.040,-178.793,5.517,148.603
C01270=1223.321,71.297,-46.056,-178.791,5.518,148.603
C01271=1223.316,71.546,-46.074,-178.788,5.519,148.602
C01272=1223.311,71.795,-46.092,-178.785,5.519,148.601
C01273=1223.307,72.045,-46.109,-178.783,5.520,148.601
C01274=1223.302,72.294,-46.127,-178.781,5.521,148.600
C01275=1223.296,72.544,-46.144,-178.778,5.521,148.600
C01276=1223.292,72.793,-46.162,-178.775,5.523,148.599
C01277=1223.287,73.042,-46.179,-178.772,5.523,148.598
C01278=1223.282,73.291,-46.197,-178.770,5.524,148.598
C01279=1223.277,73.541,-46.214,-178.767,5.525,148.597
C01280=1223.272,73.790,-46.232,-178.765,5.525,148.597
C01281=1223.268,74.040,-46.248,-178.762,5.526,148.596
C01282=1223.263,74.289,-46.266,-178.760,5.527,148.595
C01283=1223.258,74.538,-46.284,-178.757,5.528,148.595
C01284=1223.253,74.788,-46.302,-178.755,5.528,148.594
C01285=1223.248,75.037,-46.319,-178.752,5.529,148.594
C01286=1223.243,75.286,-46.337,-178.750,5.529,148.593
C01287=1223.238,75.536,-46.354,-178.747,5.530,148.593
C01288=1223.233,75.785,-46.372,-178.745,5.531,148.592
C01289=1223.228,76.035,-46.390,-178.742,5.532,148.591
C01290=1223.224,76.284,-46.407,-178.739,5.533,148.591
C01291=1223.219,76.533,-46.425,-178.737,5.534,148.590
C01292=1223.214,76.783,-46.442,-178.734,5.534,148.589
C01293=1223.209,77.032,-46.460,-178.732,5.535,148.589
C01294=1223.204,77.281,-46.478,-178.729,5.536,148.588
C01295=1223.199,77.530,-46.496,-178.727,5.536,148.588
C01296=1223.195,77.780,-46.513,-178.724,5.537,148.587
C01297=1223.190,78.029,-46.531,-178.722,5.538,148.586
C01298=1223.185,78.278,-46.549,-178.719,5.538,148.586
C01299=1223.180,78.528,-46.566,-178.717,5.539,148.585
C01300=1223.175,78.777,-46.584,-178.714,5.540,148.585
C01301=1223.170,79.026,-46.602,-178.711,5.541,148.584
C01302=1223.165,79.275,-46.620,-178.708,5.542,148.583
C01303=1223.160,79.525,-46.638,-178.706,5.543,148.583
C01304=1223.155,79.774,-46.655,-178.704,5.543,148.582
C01305=1223.150,80.023,-46.673,-178.701,5.544,148.582
C01306=1223.146,80.272,-46.691,-178.698,5.544,148.581
C01307=1223.141,80.522,-46.709,-178.696,5.545,148.581
C01308=1223.136,80.771,-46.727,-178.694,5.546,148.580
C01309=1223.131,81.021,-46.744,-178.691,5.547,148.579
C01310=1223.125,81.289,-46.763,-178.688,5.548,148.579
C01311=1223.120,81.557,-46.783,-178.685,5.549,148.578
C01312=1223.115,81.825,-46.802,-178.682,5.549,148.577
C01313=1223.110,82.094,-46.821,-178.680,5.550,148.577
C01314=1223.105,82.343,-46.839,-178.677,5.552,148.576
C01315=1223.101,82.593,-46.857,-178.675,5.552,148.576
C01316=1223.096,82.842,-46.875,-178.672,5.553,148.575
C01317=1223.091,83.092,-46.893,-178.669,5.553,148.574
C01318=1223.086,83.341,-46.911,-178.667,5.554,148.574
C01319=1223.081,83.590,-46.929,-178.665,5.555,148.573
C01320=1223.076,83.839,-46.947,-178.662,5.555,148.572
C01321=1223.071,84.088,-46.965,-178.660,5.556,148.572
C01322=1223.066,84.337,-46.983,-178.657,5.558,148.571
C01323=1223.061,84.587,-47.001,-178.654,5.558,148.571
C01324=1223.057,84.837,-47.019,-178.651,5.559,148.570
C01325=1223.052,85.086,-47.037,-178.649,5.560,148.570
C01326=1223.047,85.336,-47.054,-178.647,5.561,148.569
C01327=1223.042,85.585,-47.072,-178.644,5.561,148.568
C01328=1223.037,85.834,-47.090,-178.642,5.562,148.568
C01329=1223.031,86.083,-47.109,-178.639,5.563,148.567
C01330=1223.027,86.333,-47.128,-178.636,5.564,148.567
C01331=1223.023,86.582,-47.146,-178.633,5.565,148.566
C01332=1223.018,86.831,-47.164,-178.631,5.566,148.566
C01333=1223.013,87.080,-47.182,-178.629,5.566,148.565
C01334=1223.008,87.329,-47.200,-178.626,5.567,148.564
C01335=1223.003,87.578,-47.218,-178.624,5.568,148.564
C01336=1222.999,87.828,-47.236,-178.621,5.568,148.563
C01337=1222.994,88.078,-47.254,-178.618,5.570,148.563
C01338=1222.989,88.327,-47.272,-178.615,5.570,148.562
C01339=1222.984,88.576,-47.290,-178.613,5.571,148.561
C01340=1222.978,88.825,-47.309,-178.611,5.572,148.561
C01341=1222.974,89.075,-47.327,-178.608,5.572,148.560
C01342=1222.969,89.324,-47.345,-178.606,5.573,148.560
C01343=1222.964,89.573,-47.364,-178.603,5.574,148.559
C01344=1222.959,89.822,-47.382,-178.600,5.575,148.558
C01345=1222.955,90.071,-47.400,-178.598,5.576,148.558
C01346=1222.950,90.321,-47.418,-178.595,5.577,148.557
C01347=1222.945,90.571,-47.437,-178.593,5.578,148.557
C01348=1222.940,90.820,-47.455,-178.590,5.578,148.556
C01349=1222.935,91.068,-47.473,-178.588,5.579,148.556
C01350=1222.931,91.318,-47.492,-178.585,5.581,148.555
C01351=1222.926,91.567,-47.510,-178.582,5.581,148.554
C01352=1222.920,91.817,-47.528,-178.580,5.582,148.554
C01353=1222.915,92.066,-47.546,-178.577,5.583,148.553
C01354=1222.911,92.315,-47.565,-178.575,5.583,148.553
C01355=1222.906,92.565,-47.583,-178.573,5.584,148.552
C01356=1222.901,92.814,-47.601,-178.570,5.586,148.552
C01357=1222.896,93.063,-47.620,-178.567,5.586,148.551
C01358=1222.892,93.312,-47.639,-178.565,5.587,148.551
C01359=1222.887,93.562,-47.657,-178.562,5.588,148.550
C01360=1222.882,93.811,-47.675,-178.560,5.588,148.549
C01361=1222.877,94.061,-47.694,-178.557,5.589,148.549
C01362=1222.872,94.310,-47.713,-178.554,5.591,148.548
C01363=1222.867,94.559,-47.731,-178.552,5.591,148.547
C01364=1222.862,94.808,-47.749,-178.549,5.592,148.547
C01365=1222.858,95.058,-47.768,-178.547,5.593,148.546
C01366=1222.853,95.307,-47.786,-178.544,5.594,148.546
C01367=1222.848,95.556,-47.804,-178.542,5.595,148.545
C01368=1222.843,95.805,-47.824,-178.539,5.596,148.545
C01369=1222.838,96.055,-47.842,-178.536,5.596,148.544
C01370=1222.834,96.303,-47.860,-178.534,5.597,148.544
C01371=1222.829,96.553,-47.879,-178.532,5.598,148.543
C01372=1222.824,96.803,-47.897,-178.529,5.599,148.542
C01373=1222.819,97.051,-47.916,-178.526,5.600,148.542
C01374=1222.815,97.301,-47.934,-178.524,5.601,148.541
C01375=1222.809,97.550,-47.954,-178.521,5.602,148.541
C01376=1222.805,97.799,-47.972,-178.519,5.603,148.540
C01377=1222.799,98.049,-47.991,-178.516,5.603,148.540
C01378=1222.795,98.298,-48.009,-178.513,5.605,148.539
C01379=1222.790,98.547,-48.027,-178.511,5.606,148.539
C01380=1222.785,98.796,-48.047,-178.508,5.606,148.538
C01381=1222.780,99.046,-48.065,-178.506,5.607,148.537
C01382=1222.776,99.294,-48.084,-178.504,5.608,148.537
C01383=1222.771,99.544,-48.103,-178.500,5.609,148.536
C01384=1222.766,99.793,-48.121,-178.498,5.610,148.536
C01385=1222.761,100.043,-48.140,-178.496,5.611,148.535
C01386=1222.756,100.292,-48.159,-178.493,5.611,148.534
C01387=1222.751,100.541,-48.177,-178.490,5.613,148.534
C01388=1222.747,100.790,-48.197,-178.488,5.614,148.533
C01389=1222.742,101.040,-48.215,-178.485,5.614,148.533
C01390=1222.736,101.288,-48.234,-178.482,5.615,148.532
C01391=1222.732,101.538,-48.252,-178.480,5.616,148.532
C01392=1222.727,101.787,-48.271,-178.477,5.617,148.531
C01393=1222.723,102.036,-48.291,-178.475,5.618,148.531
C01394=1222.718,102.286,-48.308,-178.472,5.619,148.530
C01395=1222.713,102.535,-48.328,-178.470,5.619,148.529
C01396=1222.708,102.784,-48.346,-178.468,5.620,148.529
C01397=1222.703,103.033,-48.365,-178.465,5.622,148.528
C01398=1222.699,103.283,-48.384,-178.462,5.622,148.528
C01399=1222.693,103.532,-48.403,-178.460,5.623,148.527
C01400=1222.689,103.781,-48.422,-178.457,5.624,148.527
C01401=1222.684,104.030,-48.441,-178.454,5.625,148.526
C01402=1222.680,104.280,-48.460,-178.452,5.626,148.526
C01403=1222.674,104.529,-48.479,-178.449,5.627,148.525
C01404=1222.670,104.777,-48.498,-178.447,5.628,148.524
C01405=1222.665,105.028,-48.517,-178.444,5.629,148.524
C01406=1222.659,105.277,-48.536,-178.441,5.630,148.523
C01407=1222.655,105.526,-48.555,-178.439,5.631,148.523
C01408=1222.650,105.775,-48.574,-178.437,5.632,148.522
C01409=1222.646,106.025,-48.593,-178.433,5.633,148.522
C01410=1222.640,106.273,-48.612,-178.431,5.634,148.521
C01411=1222.636,106.523,-48.631,-178.429,5.635,148.520
C01412=1222.631,106.772,-48.650,-178.427,5.636,148.520
C01413=1222.627,107.021,-48.669,-178.423,5.637,148.519
C01414=1222.621,107.289,-48.689,-178.421,5.638,148.519
C01415=1222.616,107.558,-48.710,-178.418,5.638,148.518
C01416=1222.610,107.827,-48.730,-178.415,5.640,148.518
C01417=1222.605,108.095,-48.752,-178.413,5.641,148.517
C01418=1222.601,108.344,-48.770,-178.410,5.641,148.516
C01419=1222.596,108.593,-48.790,-178.408,5.643,148.516
C01420=1222.590,108.843,-48.808,-178.405,5.644,148.515
C01421=1222.586,109.092,-48.828,-178.402,5.644,148.515
C01422=1222.581,109.341,-48.847,-178.400,5.646,148.514
C01423=1222.577,109.590,-48.866,-178.397,5.647,148.514
C01424=1222.572,109.839,-48.885,-178.395,5.648,148.513
C01425=1222.567,110.089,-48.905,-178.392,5.648,148.513
C01426=1222.563,110.338,-48.924,-178.389,5.650,148.512
C01427=1222.557,110.587,-48.942,-178.387,5.651,148.512
C01428=1222.553,110.837,-48.962,-178.384,5.651,148.511
C01429=1222.548,111.085,-48.981,-178.382,5.652,148.511
C01430=1222.543,111.335,-49.000,-178.379,5.654,148.510
C01431=1222.538,111.584,-49.020,-178.376,5.654,148.509
C01432=1222.533,111.833,-49.039,-178.374,5.655,148.509
C01433=1222.529,112.082,-49.058,-178.372,5.656,148.508
C01434=1222.524,112.332,-49.078,-178.369,5.658,148.508
C01435=1222.519,112.581,-49.097,-178.366,5.658,148.507
C01436=1222.514,112.830,-49.116,-178.364,5.659,148.507
C01437=1222.510,113.079,-49.136,-178.361,5.661,148.506
C01438=1222.504,113.328,-49.155,-178.358,5.661,148.506
C01439=1222.500,113.578,-49.175,-178.356,5.662,148.505
C01440=1222.496,113.827,-49.194,-178.354,5.663,148.504
C01441=1222.490,114.076,-49.213,-178.351,5.665,148.504
C01442=1222.486,114.325,-49.233,-178.348,5.665,148.503
C01443=1222.480,114.574,-49.252,-178.346,5.666,148.503
C01444=1222.475,114.824,-49.272,-178.343,5.668,148.502
C01445=1222.471,115.073,-49.291,-178.341,5.668,148.502
C01446=1222.466,115.322,-49.310,-178.338,5.669,148.501
C01447=1222.461,115.572,-49.330,-178.336,5.670,148.501
C01448=1222.457,115.821,-49.349,-178.333,5.672,148.500
C01449=1222.451,116.070,-49.369,-178.331,5.672,148.500
C01450=1222.448,116.319,-49.388,-178.328,5.673,148.499
C01451=1222.442,116.567,-49.408,-178.325,5.675,148.499
C01452=1222.437,116.817,-49.427,-178.323,5.675,148.498
C01453=1222.433,117.067,-49.447,-178.321,5.676,148.498
C01454=1222.427,117.316,-49.466,-178.317,5.678,148.497
C01455=1222.423,117.565,-49.486,-178.315,5.679,148.497
C01456=1222.419,117.814,-49.505,-178.313,5.679,148.496
C01457=1222.414,118.063,-49.525,-178.309,5.681,148.495
C01458=1222.409,118.312,-49.545,-178.307,5.682,148.495
C01459=1222.404,118.562,-49.564,-178.305,5.682,148.494
C01460=1222.399,118.811,-49.584,-178.303,5.683,148.494
C01461=1222.394,119.060,-49.603,-178.299,5.685,148.493
C01462=1222.390,119.309,-49.624,-178.297,5.686,148.493
C01463=1222.384,119.558,-49.643,-178.295,5.686,148.492
C01464=1222.380,119.807,-49.662,-178.292,5.688,148.492
C01465=1222.375,120.057,-49.682,-178.289,5.689,148.491
C01466=1222.371,120.306,-49.702,-178.287,5.690,148.491
C01467=1222.366,120.555,-49.721,-178.284,5.691,148.490
C01468=1222.361,120.804,-49.741,-178.281,5.692,148.489
C01469=1222.356,121.054,-49.761,-178.279,5.693,148.489
C01470=1222.351,121.302,-49.781,-178.276,5.694,148.488
C01471=1222.346,121.552,-49.800,-178.274,5.695,148.488
C01472=1222.342,121.801,-49.820,-178.271,5.696,148.487
C01473=1222.337,122.050,-49.840,-178.269,5.697,148.487
C01474=1222.332,122.299,-49.860,-178.266,5.698,148.486
C01475=1222.327,122.549,-49.879,-178.264,5.699,148.486
C01476=1222.323,122.797,-49.900,-178.261,5.700,148.485
C01477=1222.318,123.047,-49.919,-178.259,5.701,148.485
C01478=1222.313,123.296,-49.939,-178.256,5.702,148.484
C01479=1222.308,123.545,-49.959,-178.253,5.704,148.484
C01480=1222.303,123.794,-49.979,-178.251,5.704,148.483
C01481=1222.299,124.043,-49.999,-178.248,5.705,148.483
C01482=1222.294,124.292,-50.018,-178.246,5.707,148.482
C01483=1222.289,124.542,-50.038,-178.243,5.707,148.482
C01484=1222.285,124.791,-50.058,-178.241,5.708,148.481
C01485=1222.280,125.040,-50.078,-178.238,5.710,148.481
C01486=1222.275,125.289,-50.098,-178.236,5.711,148.480
C01487=1222.270,125.538,-50.118,-178.232,5.712,148.480
C01488=1222.266,125.787,-50.138,-178.230,5.713,148.479
C01489=1222.261,126.037,-50.158,-178.228,5.714,148.478
C01490=1222.256,126.286,-50.178,-178.225,5.716,148.478
C01491=1222.252,126.535,-50.198,-178.222,5.716,148.477
C01492=1222.247,126.783,-50.218,-178.220,5.717,148.477
C01493=1222.242,127.033,-50.237,-178.217,5.719,148.476
C01494=1222.237,127.282,-50.258,-178.215,5.720,148.476
C01495=1222.232,127.532,-50.278,-178.212,5.720,148.475
C01496=1222.227,127.781,-50.298,-178.210,5.722,148.475
C01497=1222.223,128.030,-50.318,-178.207,5.723,148.474
C01498=1222.218,128.279,-50.338,-178.205,5.724,148.474
C01499=1222.213,128.528,-50.358,-178.202,5.725,148.473
C01500=1222.209,128.777,-50.378,-178.200,5.726,148.473
C01501=1222.204,129.026,-50.398,-178.197,5.728,148.472
C01502=1222.199,129.276,-50.419,-178.194,5.729,148.472
C01503=1222.194,129.525,-50.439,-178.192,5.729,148.471
C01504=1222.189,129.774,-50.459,-178.189,5.731,148.471
C01505=1222.184,130.023,-50.479,-178.187,5.732,148.470
C01506=1222.180,130.272,-50.499,-178.184,5.733,148.470
C01507=1222.175,130.521,-50.519,-178.181,5.734,148.469
C01508=1222.170,130.770,-50.540,-178.179,5.735,148.469
C01509=1222.166,131.019,-50.560,-178.176,5.737,148.468
C01510=1222.161,131.269,-50.580,-178.174,5.737,148.468
C01511=1222.156,131.518,-50.600,-178.171,5.738,148.467
C01512=1222.152,131.767,-50.620,-178.169,5.740,148.467
C01513=1222.146,132.017,-50.641,-178.166,5.741,148.466
C01514=1222.141,132.265,-50.661,-178.163,5.742,148.466
C01515=1222.137,132.514,-50.681,-178.161,5.743,148.465
C01516=1222.132,132.764,-50.701,-178.159,5.744,148.465
C01517=1222.127,133.013,-50.722,-178.155,5.745,148.464
C01518=1222.123,133.281,-50.744,-178.153,5.746,148.464
C01519=1222.117,133.550,-50.766,-178.150,5.748,148.463
C01520=1222.112,133.819,-50.788,-178.147,5.749,148.463
C01521=1222.107,134.087,-50.809,-178.145,5.750,148.462
C01522=1222.102,134.337,-50.830,-178.142,5.752,148.461
C01523=1222.098,134.586,-50.850,-178.140,5.753,148.461
C01524=1222.093,134.835,-50.871,-178.137,5.753,148.460
C01525=1222.089,135.084,-50.891,-178.134,5.755,148.460
C01526=1222.083,135.333,-50.911,-178.132,5.756,148.459
C01527=1222.079,135.582,-50.932,-178.129,5.758,148.459
C01528=1222.074,135.831,-50.952,-178.127,5.759,148.459
C01529=1222.069,136.081,-50.973,-178.124,5.759,148.458
C01530=1222.065,136.330,-50.993,-178.122,5.761,148.458
C01531=1222.060,136.578,-51.013,-178.119,5.762,148.457
C01532=1222.055,136.827,-51.034,-178.116,5.763,148.457
C01533=1222.050,137.077,-51.054,-178.114,5.764,148.456
C01534=1222.045,137.326,-51.074,-178.111,5.766,148.456
C01535=1222.040,137.575,-51.095,-178.109,5.766,148.455
C01536=1222.036,137.824,-51.116,-178.106,5.767,148.455
C01537=1222.031,138.073,-51.137,-178.103,5.769,148.454
C01538=1222.026,138.322,-51.157,-178.101,5.770,148.454
C01539=1222.022,138.571,-51.178,-178.098,5.772,148.453
C01540=1222.017,138.820,-51.198,-178.096,5.772,148.453
C01541=1222.012,139.069,-51.219,-178.093,5.774,148.452
C01542=1222.007,139.319,-51.240,-178.091,5.775,148.452
C01543=1222.003,139.568,-51.261,-178.088,5.776,148.451
C01544=1221.999,139.817,-51.281,-178.085,5.777,148.451
C01545=1221.993,140.066,-51.302,-178.083,5.778,148.450
C01546=1221.989,140.315,-51.322,-178.081,5.780,148.450
C01547=1221.984,140.564,-51.343,-178.078,5.781,148.449
C01548=1221.979,140.813,-51.364,-178.075,5.782,148.449
C01549=1221.974,141.063,-51.385,-178.073,5.783,148.448
C01550=1221.970,141.312,-51.405,-178.070,5.785,148.448
C01551=1221.965,141.561,-51.426,-178.067,5.786,148.447
C01552=1221.960,141.810,-51.446,-178.065,5.786,148.447
C01553=1221.955,142.059,-51.467,-178.063,5.788,148.446
C01554=1221.951,142.308,-51.488,-178.060,5.789,148.446
C01555=1221.946,142.557,-51.509,-178.057,5.791,148.445
C01556=1221.941,142.806,-51.530,-178.055,5.791,148.445
C01557=1221.936,143.055,-51.551,-178.052,5.793,148.444
C01558=1221.932,143.304,-51.571,-178.049,5.794,148.444
C01559=1221.927,143.554,-51.592,-178.047,5.796,148.443
C01560=1221.923,143.803,-51.613,-178.045,5.797,148.443
C01561=1221.917,144.052,-51.634,-178.042,5.798,148.442
C01562=1221.913,144.300,-51.655,-178.039,5.799,148.442
C01563=1221.908,144.550,-51.676,-178.036,5.801,148.441
C01564=1221.904,144.799,-51.696,-178.034,5.802,148.441
C01565=1221.899,145.048,-51.717,-178.032,5.802,148.441
C01566=1221.894,145.297,-51.737,-178.029,5.804,148.440
C01567=1221.889,145.545,-51.759,-178.027,5.805,148.440
C01568=1221.885,145.795,-51.780,-178.024,5.806,148.439
C01569=1221.880,146.044,-51.801,-178.022,5.807,148.439
C01570=1221.875,146.294,-51.822,-178.019,5.809,148.438
C01571=1221.871,146.542,-51.843,-178.016,5.810,148.438
C01572=1221.866,146.791,-51.864,-178.014,5.812,148.437
C01573=1221.861,147.040,-51.885,-178.011,5.812,148.437
C01574=1221.856,147.289,-51.905,-178.008,5.814,148.436
C01575=1221.852,147.539,-51.927,-178.006,5.815,148.436
C01576=1221.847,147.788,-51.948,-178.003,5.817,148.435
C01577=1221.842,148.037,-51.969,-178.001,5.818,148.435
C01578=1221.837,148.286,-51.990,-177.998,5.819,148.434
C01579=1221.833,148.535,-52.011,-177.996,5.820,148.434
C01580=1221.828,148.784,-52.032,-177.993,5.822,148.433
C01581=1221.823,149.033,-52.054,-177.990,5.822,148.433
C01582=1221.818,149.282,-52.075,-177.988,5.824,148.432
C01583=1221.814,149.531,-52.096,-177.985,5.825,148.432
C01584=1221.809,149.780,-52.117,-177.982,5.827,148.431
C01585=1221.804,150.029,-52.138,-177.980,5.828,148.431
C01586=1221.800,150.278,-52.159,-177.977,5.829,148.430
C01587=1221.795,150.528,-52.180,-177.975,5.830,148.430
C01588=1221.790,150.776,-52.202,-177.972,5.832,148.430
C01589=1221.786,151.025,-52.222,-177.970,5.833,148.429
C01590=1221.781,151.275,-52.243,-177.967,5.834,148.429
C01591=1221.776,151.524,-52.265,-177.965,5.835,148.428
C01592=1221.771,151.773,-52.286,-177.962,5.837,148.428
C01593=1221.767,152.021,-52.307,-177.960,5.838,148.427
C01594=1221.762,152.271,-52.328,-177.957,5.839,148.427
C01595=1221.758,152.520,-52.350,-177.955,5.840,148.426
C01596=1221.752,152.769,-52.371,-177.952,5.842,148.426
C01597=1221.748,153.018,-52.393,-177.949,5.843,148.425
C01598=1221.743,153.267,-52.413,-177.947,5.845,148.425
C01599=1221.739,153.516,-52.435,-177.945,5.846,148.424
C01600=1221.734,153.765,-52.456,-177.941,5.847,148.424
C01601=1221.729,154.014,-52.478,-177.939,5.848,148.423
C01602=1221.724,154.263,-52.500,-177.937,5.850,148.423
C01603=1221.720,154.512,-52.520,-177.934,5.850,148.422
C01604=1221.715,154.761,-52.542,-177.931,5.852,148.422
C01605=1221.710,155.010,-52.563,-177.928,5.854,148.422
C01606=1221.706,155.260,-52.585,-177.926,5.855,148.421
C01607=1221.701,155.508,-52.607,-177.923,5.857,148.421
C01608=1221.696,155.757,-52.628,-177.921,5.857,148.420
C01609=1221.692,156.006,-52.649,-177.918,5.859,148.420
C01610=1221.687,156.256,-52.670,-177.916,5.860,148.419
C01611=1221.682,156.504,-52.692,-177.913,5.862,148.419
C01612=1221.677,156.753,-52.713,-177.911,5.862,148.418
C01613=1221.673,157.003,-52.735,-177.908,5.864,148.418
C01614=1221.668,157.252,-52.756,-177.906,5.865,148.417
C01615=1221.663,157.500,-52.778,-177.903,5.867,148.417
C01616=1221.659,157.750,-52.800,-177.901,5.868,148.417
C01617=1221.654,157.999,-52.821,-177.898,5.869,148.416
C01618=1221.649,158.247,-52.842,-177.895,5.871,148.416
C01619=1221.645,158.496,-52.864,-177.893,5.872,148.415
C01620=1221.640,158.746,-52.885,-177.890,5.874,148.415
C01621=1221.635,158.994,-52.907,-177.888,5.875,148.414
C01622=1221.630,159.263,-52.931,-177.885,5.876,148.414
C01623=1221.626,159.533,-52.954,-177.882,5.878,148.413
C01624=1221.620,159.802,-52.978,-177.879,5.880,148.413
C01625=1221.615,160.071,-53.002,-177.877,5.880,148.412
C01626=1221.610,160.320,-53.023,-177.874,5.882,148.412
C01627=1221.605,160.569,-53.044,-177.871,5.883,148.411
C01628=1221.601,160.818,-53.066,-177.869,5.885,148.411
C01629=1221.596,161.067,-53.088,-177.866,5.886,148.411
C01630=1221.592,161.316,-53.110,-177.863,5.887,148.410
C01631=1221.587,161.565,-53.132,-177.861,5.889,148.410
C01632=1221.582,161.814,-53.153,-177.859,5.890,148.409
C01633=1221.577,162.063,-53.175,-177.856,5.892,148.409
C01634=1221.573,162.312,-53.196,-177.853,5.892,148.408
C01635=1221.568,162.561,-53.218,-177.851,5.894,148.408
C01636=1221.563,162.810,-53.240,-177.848,5.896,148.408
C01637=1221.559,163.059,-53.262,-177.845,5.897,148.407
C01638=1221.554,163.308,-53.284,-177.843,5.898,148.407
C01639=1221.549,163.557,-53.306,-177.841,5.899,148.406
C01640=1221.545,163.806,-53.328,-177.838,5.901,148.406
C01641=1221.540,164.055,-53.349,-177.835,5.903,148.405
C01642=1221.536,164.304,-53.371,-177.833,5.904,148.405
C01643=1221.531,164.553,-53.393,-177.830,5.906,148.404
C01644=1221.527,164.802,-53.415,-177.828,5.906,148.404
C01645=1221.522,165.051,-53.437,-177.825,5.908,148.403
C01646=1221.516,165.300,-53.459,-177.822,5.910,148.403
C01647=1221.512,165.549,-53.481,-177.820,5.910,148.402
C01648=1221.507,165.798,-53.503,-177.817,5.912,148.402
C01649=1221.503,166.047,-53.525,-177.815,5.913,148.402
C01650=1221.498,166.296,-53.546,-177.812,5.915,148.401
C01651=1221.494,166.545,-53.569,-177.809,5.917,148.401
C01652=1221.489,166.794,-53.590,-177.807,5.918,148.400
C01653=1221.485,167.043,-53.612,-177.804,5.919,148.400
C01654=1221.479,167.292,-53.635,-177.802,5.920,148.399
C01655=1221.475,167.541,-53.657,-177.799,5.922,148.399
C01656=1221.470,167.790,-53.678,-177.796,5.924,148.399
C01657=1221.466,168.039,-53.700,-177.794,5.925,148.398
C01658=1221.461,168.287,-53.723,-177.791,5.926,148.398
C01659=1221.456,168.537,-53.745,-177.789,5.927,148.397
C01660=1221.451,168.785,-53.767,-177.786,5.929,148.397
C01661=1221.447,169.035,-53.789,-177.784,5.931,148.397
C01662=1221.442,169.283,-53.811,-177.781,5.932,148.396
C01663=1221.438,169.533,-53.833,-177.779,5.933,148.396
C01664=1221.432,169.782,-53.855,-177.776,5.935,148.395
C01665=1221.428,170.030,-53.878,-177.774,5.936,148.395
C01666=1221.424,170.280,-53.900,-177.771,5.938,148.394
C01667=1221.419,170.528,-53.922,-177.769,5.939,148.394
C01668=1221.414,170.778,-53.944,-177.766,5.940,148.394
C01669=1221.410,171.026,-53.967,-177.763,5.942,148.393
C01670=1221.405,171.275,-53.989,-177.761,5.943,148.393
C01671=1221.400,171.524,-54.011,-177.758,5.945,148.392
C01672=1221.395,171.774,-54.033,-177.755,5.947,148.392
C01673=1221.391,172.022,-54.055,-177.753,5.948,148.391
C01674=1221.387,172.271,-54.077,-177.750,5.949,148.391
C01675=1221.382,172.521,-54.100,-177.747,5.951,148.390
C01676=1221.377,172.769,-54.123,-177.745,5.952,148.390
C01677=1221.373,173.018,-54.145,-177.743,5.954,148.390
C01678=1221.367,173.267,-54.167,-177.740,5.954,148.389
C01679=1221.363,173.516,-54.189,-177.737,5.956,148.389
C01680=1221.359,173.765,-54.212,-177.735,5.958,148.388
C01681=1221.353,174.014,-54.234,-177.733,5.959,148.388
C01682=1221.349,174.263,-54.257,-177.730,5.961,148.387
C01683=1221.344,174.511,-54.278,-177.727,5.962,148.387
C01684=1221.339,174.761,-54.301,-177.725,5.963,148.387
C01685=1221.335,175.010,-54.324,-177.722,5.965,148.386
C01686=1221.330,175.259,-54.346,-177.719,5.967,148.386
C01687=1221.326,175.507,-54.369,-177.717,5.968,148.385
C01688=1221.322,175.757,-54.391,-177.714,5.970,148.385
C01689=1221.316,176.006,-54.413,-177.712,5.971,148.385
C01690=1221.312,176.255,-54.436,-177.709,5.972,148.384
C01691=1221.307,176.504,-54.459,-177.706,5.974,148.384
C01692=1221.303,176.752,-54.481,-177.704,5.976,148.383
C01693=1221.298,177.002,-54.504,-177.702,5.977,148.383
C01694=1221.294,177.251,-54.526,-177.699,5.978,148.383
C01695=1221.289,177.499,-54.548,-177.696,5.980,148.382
C01696=1221.284,177.748,-54.571,-177.694,5.981,148.382
C01697=1221.280,177.998,-54.593,-177.691,5.983,148.381
C01698=1221.274,178.246,-54.616,-177.688,5.985,148.381
C01699=1221.270,178.495,-54.638,-177.686,5.986,148.381
C01700=1221.265,178.744,-54.662,-177.684,5.987,148.380
C01701=1221.261,178.992,-54.684,-177.681,5.989,148.380
C01702=1221.256,179.242,-54.707,-177.678,5.990,148.379
C01703=1221.252,179.491,-54.730,-177.676,5.992,148.379
C01704=1221.246,179.740,-54.752,-177.673,5.994,148.379
C01705=1221.242,179.988,-54.775,-177.670,5.995,148.378
C01706=1221.238,180.237,-54.798,-177.668,5.996,148.378
C01707=1221.233,180.487,-54.820,-177.665,5.998,148.377
C01708=1221.228,180.735,-54.843,-177.663,6.000,148.377
C01709=1221.224,180.984,-54.865,-177.661,6.001,148.376
C01710=1221.219,181.233,-54.888,-177.658,6.003,148.376
C01711=1221.215,181.482,-54.911,-177.655,6.004,148.376
C01712=1221.210,181.731,-54.934,-177.653,6.005,148.375
C01713=1221.205,181.980,-54.957,-177.650,6.007,148.375
C01714=1221.201,182.229,-54.980,-177.647,6.009,148.374
C01715=1221.196,182.478,-55.003,-177.645,6.011,148.374
C01716=1221.191,182.727,-55.025,-177.642,6.011,148.373
C01717=1221.187,182.976,-55.048,-177.639,6.013,148.373
C01718=1221.182,183.225,-55.071,-177.637,6.015,148.373
C01719=1221.178,183.473,-55.094,-177.635,6.016,148.372
C01720=1221.172,183.722,-55.116,-177.632,6.018,148.372
C01721=1221.168,183.971,-55.139,-177.629,6.020,148.372
C01722=1221.164,184.220,-55.163,-177.626,6.021,148.371
C01723=1221.159,184.469,-55.186,-177.624,6.022,148.371
C01724=1221.155,184.718,-55.208,-177.622,6.024,148.370
C01725=1221.149,184.967,-55.231,-177.619,6.026,148.370
C01726=1221.145,185.237,-55.256,-177.616,6.028,148.370
C01727=1221.140,185.507,-55.281,-177.613,6.029,148.369
C01728=1221.135,185.776,-55.306,-177.610,6.031,148.369
C01729=1221.130,186.046,-55.332,-177.608,6.033,148.368
C01730=1221.125,186.294,-55.353,-177.605,6.033,148.368
C01731=1221.120,186.543,-55.377,-177.603,6.035,148.367
C01732=1221.116,186.792,-55.400,-177.600,6.037,148.367
C01733=1221.112,187.041,-55.423,-177.598,6.038,148.367
C01734=1221.107,187.290,-55.446,-177.595,6.040,148.366
C01735=1221.102,187.539,-55.469,-177.593,6.042,148.366
C01736=1221.097,187.787,-55.492,-177.589,6.043,148.365
C01737=1221.093,188.036,-55.515,-177.587,6.044,148.365
C01738=1221.088,188.285,-55.539,-177.585,6.046,148.365
C01739=1221.083,188.534,-55.562,-177.582,6.048,148.364
C01740=1221.079,188.783,-55.585,-177.579,6.050,148.364
C01741=1221.075,189.032,-55.608,-177.577,6.051,148.364
C01742=1221.070,189.281,-55.631,-177.575,6.053,148.363
C01743=1221.065,189.530,-55.655,-177.571,6.054,148.363
C01744=1221.060,189.778,-55.678,-177.569,6.056,148.362
C01745=1221.056,190.027,-55.701,-177.567,6.057,148.362
C01746=1221.051,190.276,-55.724,-177.564,6.059,148.362
C01747=1221.047,190.525,-55.747,-177.561,6.061,148.361
C01748=1221.042,190.774,-55.771,-177.559,6.063,148.361
C01749=1221.037,191.023,-55.794,-177.557,6.064,148.361
C01750=1221.033,191.272,-55.817,-177.554,6.065,148.360
C01751=1221.029,191.521,-55.840,-177.551,6.067,148.360
C01752=1221.024,191.770,-55.863,-177.548,6.069,148.359
C01753=1221.019,192.019,-55.887,-177.546,6.071,148.359
C01754=1221.015,192.268,-55.910,-177.544,6.072,148.359
C01755=1221.009,192.516,-55.933,-177.541,6.073,148.358
C01756=1221.005,192.765,-55.957,-177.538,6.075,148.358
C01757=1221.000,193.014,-55.981,-177.536,6.077,148.358
C01758=1220.996,193.262,-56.003,-177.534,6.078,148.357
C01759=1220.992,193.512,-56.027,-177.531,6.080,148.357
C01760=1220.987,193.761,-56.050,-177.528,6.081,148.356
C01761=1220.982,194.010,-56.073,-177.525,6.083,148.356
C01762=1220.978,194.258,-56.098,-177.522,6.085,148.356
C01763=1220.973,194.507,-56.121,-177.520,6.086,148.355
C01764=1220.968,194.756,-56.144,-177.518,6.088,148.355
C01765=1220.964,195.005,-56.168,-177.515,6.090,148.354
C01766=1220.959,195.254,-56.192,-177.512,6.092,148.354
C01767=1220.955,195.503,-56.215,-177.510,6.093,148.354
C01768=1220.950,195.752,-56.238,-177.508,6.094,148.353
C01769=1220.945,196.001,-56.262,-177.505,6.096,148.353
C01770=1220.941,196.249,-56.286,-177.502,6.098,148.352
C01771=1220.936,196.498,-56.309,-177.499,6.100,148.352
C01772=1220.931,196.747,-56.333,-177.497,6.101,148.352
C01773=1220.927,196.996,-56.357,-177.495,6.103,148.351
C01774=1220.922,197.245,-56.380,-177.492,6.104,148.351
C01775=1220.918,197.494,-56.403,-177.489,6.106,148.351
C01776=1220.913,197.742,-56.427,-177.487,6.108,148.350
C01777=1220.908,197.991,-56.451,-177.485,6.109,148.350
C01778=1220.904,198.240,-56.474,-177.482,6.111,148.350
C01779=1220.899,198.488,-56.498,-177.479,6.113,148.349
C01780=1220.895,198.737,-56.522,-177.477,6.115,148.349
C01781=1220.890,198.987,-56.545,-177.474,6.116,148.348
C01782=1220.886,199.235,-56.569,-177.471,6.118,148.348
C01783=1220.881,199.484,-56.592,-177.469,6.119,148.348
C01784=1220.877,199.732,-56.616,-177.466,6.121,148.347
C01785=1220.872,199.981,-56.640,-177.464,6.123,148.347
C01786=1220.868,200.231,-56.664,-177.461,6.124,148.347
C01787=1220.863,200.480,-56.688,-177.458,6.126,148.346
C01788=1220.859,200.728,-56.712,-177.456,6.128,148.346
C01789=1220.853,200.977,-56.736,-177.454,6.129,148.346
C01790=1220.849,201.226,-56.760,-177.451,6.131,148.345
C01791=1220.844,201.475,-56.783,-177.448,6.133,148.345
C01792=1220.840,201.723,-56.807,-177.446,6.135,148.345
C01793=1220.835,201.972,-56.830,-177.443,6.137,148.344
C01794=1220.831,202.221,-56.855,-177.440,6.138,148.344
C01795=1220.826,202.470,-56.878,-177.438,6.139,148.344
C01796=1220.822,202.719,-56.903,-177.435,6.141,148.343
C01797=1220.817,202.968,-56.926,-177.432,6.143,148.343
C01798=1220.813,203.217,-56.950,-177.430,6.145,148.342
C01799=1220.808,203.465,-56.974,-177.427,6.146,148.342
C01800=1220.803,203.714,-56.998,-177.425,6.148,148.342
C01801=1220.799,203.962,-57.022,-177.422,6.149,148.341
C01802=1220.794,204.212,-57.046,-177.420,6.151,148.341
C01803=1220.789,204.460,-57.070,-177.417,6.153,148.341
C01804=1220.785,204.709,-57.094,-177.415,6.155,148.340
C01805=1220.781,204.958,-57.118,-177.412,6.157,148.340
C01806=1220.776,205.207,-57.142,-177.409,6.159,148.340
C01807=1220.771,205.455,-57.166,-177.407,6.160,148.339
C01808=1220.767,205.704,-57.190,-177.405,6.161,148.339
C01809=1220.762,205.953,-57.214,-177.402,6.163,148.339
C01810=1220.758,206.202,-57.238,-177.399,6.165,148.338
C01811=1220.753,206.451,-57.263,-177.397,6.167,148.338
C01812=1220.749,206.700,-57.286,-177.394,6.169,148.338
C01813=1220.744,206.948,-57.310,-177.391,6.171,148.337
C01814=1220.739,207.197,-57.335,-177.389,6.173,148.337
C01815=1220.735,207.447,-57.359,-177.387,6.174,148.336
C01816=1220.730,207.695,-57.383,-177.384,6.175,148.336
C01817=1220.726,207.943,-57.407,-177.381,6.177,148.336
C01818=1220.721,208.192,-57.432,-177.379,6.179,148.335
C01819=1220.717,208.441,-57.456,-177.376,6.181,148.335
C01820=1220.712,208.690,-57.479,-177.373,6.183,148.335
C01821=1220.707,208.939,-57.504,-177.371,6.185,148.334
C01822=1220.703,209.187,-57.528,-177.368,6.186,148.334
C01823=1220.699,209.436,-57.552,-177.366,6.187,148.334
C01824=1220.694,209.685,-57.577,-177.363,6.189,148.333
C01825=1220.690,209.934,-57.601,-177.361,6.191,148.333
